FOR mv_i := 1 TO MOVER_NUMBER BY 1 DO
    // Only check for bMoverSync when the WaitOnExternalTrigger scenario is selected
    IF __ISVALIDREF(_MoverList[mv_i].Station.Process) AND
       _MoverList[mv_i].Station.ApproachScenario = ApproachScenario_e.WaitOnExternalTrigger THEN
        //bMoverSync := bMoverSync AND
        //              (_MoverList[i].Station.Process.xMoverPathFree AND NOT _MoverList[i].Station.Process.xNeedMover);
    END_IF
END_FOR

// start update simu mover **********************************************
IF CONST.USE_SIMULATION THEN
    FOR mv_i := 1 TO MOVER_NUMBER BY 1 DO
        _MoverList[mv_i].MoverAxis(xIN_StopMover := HMI_xStopMover);
    END_FOR
END_IF

// stop update simu mover **********************************************

// start communication with B&R PLC ************************************
FOR mv_i := 1 TO CONST.STATION_NUMBER BY 1 DO
    IF __ISVALIDREF(_MoverList[mv_i].Station) AND __ISVALIDREF(_20_AUTO.recipe) THEN
        _StationList[mv_i].Offset := _20_AUTO.recipe.stationOffsets[mv_i - 1];
    END_IF
END_FOR

IF CONST.BIND_WITH_TRACK AND gMoverAxis.Q_CT_Track_to_BR.asStruct.bCommand.enableProcess THEN
    FOR mv_i := 1 TO MOVER_NUMBER BY 1 DO
        IF __ISVALIDREF(_MoverList[mv_i].Station) THEN
            gMoverAxis.Q_CT_Shuttle_to_BR.asStruct[mv_i].bCommand.release :=
                ((THIS^._MoverList[mv_i].State = MoverState_e.WaitLeaveCurrentStation) OR
                (_MoverList[mv_i].State = MoverState_e.MovingToStation) OR
                (_MoverList[mv_i].State = MoverState_e.PerformRelativeMove)) AND
                gMoverAxis.I_CT_Shuttle_from_BR.asStruct[mv_i].bStatus.at_target;

            gMoverAxis.Q_CT_Shuttle_to_BR.asStruct[mv_i].bNextStation    := _MoverList[mv_i].Station.SuperTrackNumber;
            gMoverAxis.Q_CT_Shuttle_to_BR.asStruct[mv_i].diNextOffset_um :=
                LREAL_TO_DINT(_MoverList[mv_i].Station.Offset * 1000.0 +
                              _MoverList[mv_i].MovingProcessOffset * 1000.0);

            // echo At_Target
            gMoverAxis.Q_CT_Shuttle_to_BR.asStruct[mv_i].bCommand.echo_At_Target :=
                gMoverAxis.I_CT_Shuttle_from_BR.asStruct[mv_i].bStatus.at_target;

            // echo at position
            gMoverAxis.Q_CT_Shuttle_to_BR.asStruct[mv_i].bCommand.echo_in_pos :=
                gMoverAxis.I_CT_Shuttle_from_BR.asStruct[mv_i].bStatus.in_position;

            // Quit
            gMoverAxis.Q_CT_Track_to_BR.asStruct.bCommand.resetErrors := HMI.btArMain[7].press;
        END_IF
    END_FOR
END_IF

// stop communication with B&R PLC ************************************

// test if path is free
IF CONST.BIND_WITH_TRACK THEN
    gMoverAxis.Q_CT_Track_to_BR.asStruct.bCommand.wholePathFree := TRUE;

    FOR mv_i := 1 TO CONST.STATION_NUMBER BY 1 DO
        IF __ISVALIDREF(_StationList[mv_i].Process) AND_THEN NOT _StationList[mv_i].Process.xMoverPathFree THEN
            gMoverAxis.Q_CT_Track_to_BR.asStruct.bCommand.wholePathFree := FALSE;
        END_IF
    END_FOR

    IF HMI.enState = enState.StateMANU THEN
        gMoverAxis.Q_CT_Track_to_BR.asStruct.bCommand.wholePathFree := TRUE;
    END_IF
END_IF

// start collision check **********************************************
IF NOT CONST.BIND_WITH_TRACK THEN
    FOR mv_i := 1 TO MOVER_NUMBER - 1 BY 1 DO
        _MoverList[mv_i].MoverAxis.IsColliding(_MoverList[mv_i + 1].MoverAxis);
        _MoverList[mv_i].MoverAxis.WillCollide(_MoverList[mv_i + 1].MoverAxis);

        IF THIS^.IsMoverLost(THIS^._MoverList[mv_i]) THEN
            // ASSERT HERE, WE SHOULD NEVER GO HERE
            ASSERT(0);
        END_IF
    END_FOR

    _MoverList[MOVER_NUMBER].MoverAxis.IsColliding(_MoverList[1].MoverAxis); // do not forget to test this case, too
    _MoverList[MOVER_NUMBER].MoverAxis.WillCollide(_MoverList[1].MoverAxis);
END_IF

// end collision check **********************************************

// start output affectation **********************************************
xOUT_AllMoverEmpty := TRUE;

FOR mv_i := 1 TO MOVER_NUMBER BY 1 DO
    IF _MoverList[mv_i].GetLastStationDone() <> 0 THEN
        xOUT_AllMoverEmpty := FALSE;
    END_IF
END_FOR

xOUT_Error := gMoverAxis.I_CT_Track_from_BR.asStruct.bStatus.error;

// end output affectation **********************************************

// This method check if the wait pos of a given station is before another
// station. This situation is not permitted by the system, yet
METHOD CheckWaitPosNotBehindStation : BOOL
VAR_INPUT
END_VAR
VAR
    i : INT;
END_VAR
CheckWaitPosNotBehindStation := FALSE;
FOR i := 2 TO CONST.STATION_NUMBER BY 1 DO
    CheckWaitPosNotBehindStation := CheckWaitPosNotBehindStation OR
        THIS^._StationList[i].Position.lrWorkPosition + THIS^._StationList[i].WaitPos <
        THIS^._StationList[i - 1].Position.lrWorkPosition;
END_FOR

// NO CHECK ARE MADE BETWEEN THE FIRST POS AND THE LAST
END_METHOD

METHOD Equals : BOOL
VAR_INPUT
    object : ANY;
END_VAR
Equals := THIS = object.pValue;
END_METHOD

METHOD FB_init : BOOL
VAR_INPUT
    bInitRetains : BOOL; // if TRUE, the retain variables are initialized (warm start / cold start)
    bInCopyCode  : BOOL; // if TRUE, the instance afterwards gets moved into the copy code (online change)
END_VAR
VAR
    i : INT;
END_VAR
THIS^._iID := THIS^._iInstanceCounter;
THIS^._iInstanceCounter := THIS^._iInstanceCounter +1;
END_METHOD

METHOD GetMoverIndex : INT
VAR_INPUT
    mover : REFERENCE TO FB_Mover;
END_VAR
VAR
    i : INT;
END_VAR
FOR i:= 1 TO THIS^.MOVER_NUMBER BY 1 DO 
	IF mover.Equals(THIS^._MoverList[i]) THEN
		GetMoverIndex := i;
		EXIT;
	END_IF
END_FOR
END_METHOD

// Get the mover with the next number (Means the mover behind)
METHOD GetNextMover : REFERENCE TO FB_Mover
VAR_INPUT
    Mover : REFERENCE TO FB_Mover;
END_VAR
VAR
    moverIndex : INT;
END_VAR
moverIndex := THIS^.GetMoverIndex(Mover);

IF moverIndex >= THIS^.MOVER_NUMBER THEN
    GetNextMover REF= THIS^._MoverList[1];
ELSE
    GetNextMover REF= THIS^._MoverList[moverIndex + 1];
END_IF
END_METHOD

// we check if there is a mover between refMover and the refMover.Station
// This method is used to unblock a mover that cannot move because of a mover
// "Behind" it that also want to move to the same station
METHOD PRIVATE GetNumOfMoverOnTheWay : INT
VAR_INPUT
    refMover : REFERENCE TO FB_Mover; // The maybe stucking mover
END_VAR
VAR
    lrMoverPosTemp   : LREAL; // we use this position beacuse maybe we are at the end of the track
    lrStationPosTemp : LREAL; // we use this position beacuse maybe we are at the end of the track
    i                : INT;
END_VAR
GetNumOfMoverOnTheWay := 0;

FOR i := 1 TO THIS^.MOVER_NUMBER BY 1 DO
    // If the mover is in front of the tested mover, we add MAX_TRACK_LENGTH (maybe we are at the end of the track ?)
    IF refMover.IsInFront(THIS^._MoverList[i].MoverAxis.CurrentPos) THEN
        lrMoverPosTemp := THIS^._MoverList[i].MoverAxis.CurrentPos + CONST.MAX_TRACK_LENGTH;
    ELSE
        lrMoverPosTemp := THIS^._MoverList[i].MoverAxis.CurrentPos;
    END_IF

    // If the mover is in front of the station, we add MAX_TRACK_LENGTH (maybe we are at the end of the track ?)
    IF refMover.IsInFront(refMover.Station.Position.lrWorkPosition) THEN
        lrStationPosTemp := refMover.Station.Position.lrWorkPosition + CONST.MAX_TRACK_LENGTH;
    ELSE
        lrStationPosTemp := refMover.Station.Position.lrWorkPosition;
    END_IF

    IF (lrMoverPosTemp > refMover.MoverAxis.CurrentPos) AND
       (lrMoverPosTemp <= lrStationPosTemp + refMover.AttachedPieceHolder.PosOffset) THEN
	   // If a mover is at position but has
        GetNumOfMoverOnTheWay := GetNumOfMoverOnTheWay + 1;
    END_IF
END_FOR
END_METHOD

// Get the mover with the previous number (Means the front mover)
METHOD GetPrevMover : REFERENCE TO FB_Mover
VAR_INPUT
    Mover : REFERENCE TO FB_Mover;
END_VAR
VAR
    moverIndex : INT;
END_VAR
moverIndex := THIS^.GetMoverIndex(Mover);

IF moverIndex <= 1 THEN
    GetPrevMover REF= THIS^._MoverList[THIS^.MOVER_NUMBER];
ELSE
    GetPrevMover REF= THIS^._MoverList[moverIndex - 1];
END_IF
END_METHOD

METHOD IsAllMoverAtPosition : BOOL
VAR_INPUT
END_VAR
VAR
    i : INT;
END_VAR
IsAllMoverAtPosition := TRUE;

FOR i := 1 TO THIS^.MOVER_NUMBER BY 1 DO
    IF (THIS^._MoverList[i].State = MoverState_e.WaitLeaveCurrentStation) OR
       (THIS^._MoverList[i].State = MoverState_e.MovingToStation) OR
       (THIS^._MoverList[i].State = MoverState_e.InStationPos) THEN
        IsAllMoverAtPosition := FALSE;
        EXIT;
    END_IF
END_FOR
END_METHOD

// Is a shuttle present in the given region?
// If 'from_pos' is greater than 'to_pos', this means we look in
// a region that include the begining of the track
METHOD PUBLIC IsMoverInRange : BOOL
VAR_INPUT
    from_pos : LREAL; // begin of the tested region (included)
    to_pos   : LREAL; // end of the tested region (included)
END_VAR
VAR
    i       : INT;
END_VAR

IsMoverInRange := FALSE;

IF from_pos < to_pos THEN
    FOR i := 1 TO THIS^.MOVER_NUMBER BY 1 DO
        IF (THIS^._MoverList[i].MoverAxis.CurrentPos >= from_pos) AND
           (THIS^._MoverList[i].MoverAxis.CurrentPos <= to_pos) THEN
		   IsMoverInRange := TRUE;
		   EXIT;
		   
        END_IF
    END_FOR
ELSE // we test a region that pass by the maximum track length
    FOR i := 1 TO THIS^.MOVER_NUMBER BY 1 DO
        IF (THIS^._MoverList[i].MoverAxis.CurrentPos >= from_pos) OR
           (THIS^._MoverList[i].MoverAxis.CurrentPos <= to_pos) THEN
		   IsMoverInRange := TRUE;
		   EXIT;
		   
        END_IF
    END_FOR
END_IF
END_METHOD

// If the target station of a mover is not between the target of the previous and the next mover
// this function will return true. This function is attendend to debug only
METHOD IsMoverLost : BOOL
VAR_INPUT
    mover : REFERENCE TO FB_Mover;
END_VAR
VAR
    i : INT;

    prevStationLoc  : LREAL;
    nextStationLoc  : LREAL;
    moverStationLoc : LREAL; // mover to test location
    posList         : ARRAY[0..2] OF LREAL;
END_VAR
(* the algorithm function as fallow 

First we built a sorted array based on the station position
Then we search for the previous station position and fix
our search index
Then we check if the squence of mover is correct. The sequence must be
PreviousMoverStation -> CurrentMoverStation -> NextMoverStation
If we don't get this sequence, then the mover is lost.

In fact, since we have only 3 elements, we only need to check
the next station
*)
IsMoverLost := FALSE;

nextStationLoc  := THIS^.GetNextMover(mover).Station.Position.lrWorkPosition;
prevStationLoc  := THIS^.GetPrevMover(mover).Station.Position.lrWorkPosition;
moverStationLoc := mover.station.Position.lrWorkPosition;

posList[0] := prevStationLoc;
posList[1] := moverStationLoc;
posList[2] := nextStationLoc;

SortBubbleLREAL(ADR(posList), 0, 2);

IF posList[0] = prevStationLoc THEN
    IF posList[1] <> moverStationLoc THEN
        IsMoverLost := TRUE;
    END_IF

ELSIF posList[0] = moverStationLoc THEN
    IF posList[1] <> nextStationLoc THEN
        IsMoverLost := TRUE;
    END_IF

ELSE (* posList[0] = nextStationLoc *)
    IF posList[1] <> prevStationLoc THEN
        IsMoverLost := TRUE;
    END_IF
END_IF
END_METHOD

METHOD PRIVATE IsMoverMovingToStation : BOOL
VAR_INPUT
    iMoverNumber : INT; // the current mover number 
END_VAR
VAR
    i           : INT;
END_VAR
IsMoverMovingToStation := FALSE;

FOR i := 1 TO THIS^.MOVER_NUMBER BY 1 DO

    // we don't check the tests mover station, else it will be always true
    IF (iMoverNumber <> i) AND THIS^._MoverList[i].Station.Equals(THIS^._MoverList[iMoverNumber].Station) THEN
        IsMoverMovingToStation := IsMoverMovingToStation OR
                                  (THIS^._MoverList[i].State = MoverState_e.WaitLeaveCurrentStation) OR
                                  (THIS^._MoverList[i].State = MoverState_e.MovingToStation) OR
                                  (THIS^._MoverList[i].State = MoverState_e.InStationPos);

        // Do not exit here, since we OR the flag
        // TODO maybe we should add an IF statement to exit when the flag is true
        // because it will never be false again ... ? // PERFORMANCE ISSUE
    END_IF

END_FOR
END_METHOD

// Return TRUE if at least one mover is stucked
METHOD IsMoverStucked : BOOL
VAR_INPUT
END_VAR
IsMoverStucked := FALSE;

FOR mv_i := 1 TO THIS^.MOVER_NUMBER BY 1 DO
    IF THIS^._MoverList[mv_i].MoverAxis.xStuck THEN
        IsMoverStucked := TRUE;
        EXIT;
    END_IF
END_FOR
END_METHOD

// Is the given process used by the current station configuration?
METHOD IsProcessUsed : BOOL
VAR_INPUT
    this_process : REFERENCE TO FB_AUT_ABSTRACT;
END_VAR
VAR
	i : INT;
END_VAR
IsProcessUsed := THIS^._WorkStationList[PH_num].IsProcessUsed(this_process);
END_METHOD

METHOD SetAllScenario : REFERENCE TO FB_MoverMan
VAR_INPUT
END_VAR
VAR
	i : INT;
END_VAR
FOR i := 1 TO CONST.STATION_NUMBER BY 1 DO
    THIS^._StationList[i].ApproachScenario := THIS^.HMI_Scenario;
END_FOR

SetAllScenario REF= THIS^;
END_METHOD

// Give a random time for each process. It ensure at least the minimum and the maximum value are given
// to at least 2 diffrents process
METHOD SetAllTimers : REFERENCE TO FB_MoverMan
VAR_INPUT
    arrStationTime : POINTER TO DINT;
    udiOffset      : UDINT; // simple offset to apply to the seed
END_VAR
VAR
    i         : INT;
    rand      : DRAND;
    tempIndex : INT := 0;
    getTime   : GETSYSTEMTIME;
END_VAR
IF arrStationTime <> 0 THEN
	
    getTime();
    rand.Seed := TO_INT(getTime.timeLoDW + udiOffset);

    FOR i := 0 TO CONST.STATION_NUMBER - 1 BY 1 DO
        rand();
        arrStationTime[i] := TO_DINT((THIS^.HMI_TimeMax - THIS^.HMI_TimeMin) * (rand.Num) + THIS^.HMI_TimeMin);
    END_FOR

    tempIndex := 0;

    FOR i := 1 TO CONST.STATION_NUMBER - 1 BY 1 DO
        IF arrStationTime[i] < arrStationTime[tempIndex] THEN
            tempIndex := i;
        END_IF
    END_FOR

    arrStationTime[tempIndex] := THIS^.HMI_TimeMin;

    tempIndex := 0;

    FOR i := 1 TO CONST.STATION_NUMBER - 1 BY 1 DO
        IF arrStationTime[i] > arrStationTime[tempIndex] THEN
            tempIndex := i;
        END_IF
    END_FOR

    arrStationTime[tempIndex] := THIS^.HMI_TimeMax;
END_IF

SetAllTimers REF= THIS^;
END_METHOD

METHOD ToString : STRING
VAR_INPUT
END_VAR
ToString := CONCAT('FB_MoverMan_', TO_STRING(THIS^._iID));
END_METHOD

END_FUNCTION_BLOCK

// ---- POUs/20_AUTO/Mover/FB_PieceHolder.TcPOU
FUNCTION_BLOCK FB_PieceHolder
VAR_INPUT
END_VAR
VAR_OUTPUT
END_VAR
VAR
	_lrPosOffset : LREAL; // current offset position
	
	_iID : INT := 0; // instance ID, is set during FB_Init using the value of _iInstanceCounter 
END_VAR
VAR_STAT
	_iInstanceCounter : INT := 1; // instance counter
END_VAR

METHOD FB_init : BOOL
VAR_INPUT
    bInitRetains : BOOL;  // if TRUE, the retain variables are initialized (warm start / cold start)
    bInCopyCode  : BOOL;  // if TRUE, the instance afterwards gets moved into the copy code (online change)
    offset       : LREAL; //position offset of the tool using this toolhead, a negative value represents a move on the left
END_VAR
THIS^._iID := THIS^._iInstanceCounter;
THIS^._iInstanceCounter := THIS^._iInstanceCounter +1;
THIS^.PosOffset := offset;
END_METHOD

PROPERTY PosOffset : LREAL
GET
PosOffset := _lrPosOffset;
END_GET
SET
_lrPosOffset := PosOffset;
END_SET
END_PROPERTY

METHOD ToString : STRING
VAR_INPUT
END_VAR
ToString := CONCAT('FB_PieceHolder_', TO_STRING(THIS^._iID));
END_METHOD

END_FUNCTION_BLOCK

// ---- POUs/20_AUTO/Mover/FB_SimuMoverAxis.TcPOU
FUNCTION_BLOCK FB_SimuMoverAxis IMPLEMENTS IObject
VAR_INPUT
    xIN_StopMover : BOOL; // stop the mover from movinf
END_VAR
VAR_OUTPUT
    outSimuCurrentPos   : Pos2D_t; // Mover position, expressed as slot number
    outSimuCurrentPosSC : Pos2D_t; // Mover position, expressed as pixel for SC
    outSimuCurrentRot   : INT;     // mover current rotation
    isInPos             : BOOL;    // true when targetPos = currentPos
END_VAR
VAR
    // with tick rate at 10ms, a value of 10 gives us 1m/s
    _Velocity    : LREAL := 0;     // Mover velocity, expressed as mm per tick, max is 10m/s
    _ErrorState  : INT   := 0;     // error state, not used
    _TargetPos   : LREAL := 0;     // last target pos
    _CurrentPos  : LREAL := 0;     // Current Pos, but with more resolution than the pixel
    _IsColliding : BOOL  := FALSE; // When true, the mover should not move
    _LastPos     : LREAL := 0;     // last position, used to trigger the xStuck flag
    _xStuck      : BOOL;           // true when the axis does not move
    _willCollide : BOOL := FALSE;  // TRUE if a collision will occure with the current velocity

    {attribute 'hide'}
    _lrNextStopPos : LREAL; // local variable used to get next stop

    _iID : INT := 0; // instance ID, is set during FB_Init using the value of _iInstanceCounter 

    _CurrentDir : MoverDirection_e := MoverDirection_e.Farward;
END_VAR

VAR_TEMP
    _MoverAccel : LREAL; // Mover acceleration, can be positive or negative depending on the direction
END_VAR

VAR CONSTANT
    MAX_POS  : LREAL := CONST.MAX_TRACK_LENGTH; // should be defined elsewhere ...
    MAX_SIZE : LREAL := CONST.MAX_MOVER_SIZE;   // Maxium size of the mover
    //MOVER_ACCEL        : LREAL := 0.1;                      // Mover acceleration, in mm/tick^2
    //MOVER_VELOCITY_MAX : LREAL := 20;                     // Mover velocity, expressed as mm per tick, max is 10m/s
    MOVER_VELOCITY_MIN : LREAL := 1; // Mover velocity, expressed as mm per tick, max is 10m/s
END_VAR
VAR_STAT
    _iInstanceCounter : INT := 1; // instance counter
END_VAR

IF NOT xIN_StopMover THEN // Do not change momemtum when we stop the movers from HMI
    IF MoverDirection_e.Farward = THIS^._CurrentDir THEN
        _MoverAccel := SIMU.lrAccelMover;
    ELSE
        _MoverAccel := -SIMU.lrAccelMover;
    END_IF

    IF NOT _IsColliding THEN

        IF THIS^.GetStopLen(_Velocity, SIMU.lrAccelMover) >= DistToTravel(_CurrentPos, _TargetPos) OR
           THIS^._willCollide THEN
            _Velocity := _Velocity - _MoverAccel;

        ELSIF SIMU.lrSpeedMover > ABS(_Velocity) AND _CurrentPos <> _TargetPos THEN
            _Velocity := _Velocity + _MoverAccel;

        END_IF
    ELSE
        _Velocity := _Velocity - _MoverAccel;
    END_IF
END_IF

// protect max and min speed
IF SIMU.lrSpeedMover < ABS(_Velocity) THEN
    IF MoverDirection_e.Farward = THIS^._CurrentDir THEN
        _Velocity := SIMU.lrSpeedMover;
    ELSE
        _Velocity := -SIMU.lrSpeedMover;
    END_IF
ELSIF ABS(_Velocity) < MOVER_VELOCITY_MIN THEN
    IF MoverDirection_e.Farward = THIS^._CurrentDir THEN
        _Velocity := MOVER_VELOCITY_MIN;
    ELSE
        _Velocity := -MOVER_VELOCITY_MIN;
    END_IF
END_IF

IF NOT _IsColliding AND NOT xIN_StopMover THEN

    IF DistToTravel(_CurrentPos, _TargetPos) > ABS(_Velocity) THEN
        _CurrentPos := _CurrentPos + _Velocity;

    ELSE
        _CurrentPos := _TargetPos;
        _Velocity   := 0;

    END_IF
END_IF

IF _CurrentPos >= MAX_POS THEN
    _CurrentPos := _CurrentPos - MAX_POS;
    // we prevent the stuck flag to be true at the end of the track
    THIS^._LastPos := THIS^._LastPos - MAX_POS;
END_IF

isInPos := EqualDelta(_CurrentPos, _TargetPos, 1.0); // we use delta comparison beacause axis is always at a low value 

outSimuCurrentPos   := THIS^.ResolvePos(THIS^.CurrentPos, outSimuCurrentRot);
outSimuCurrentPosSC := THIS^.ResolvePosSC(THIS^.CurrentPos, outSimuCurrentRot);

_xStuck        := (THIS^._CurrentPos < (THIS^._LastPos + _Velocity)) AND NOT isInPos;
THIS^._LastPos := THIS^._CurrentPos;

PROPERTY CurrentPos : LREAL
GET
IF CONST.BIND_WITH_TRACK THEN
    CurrentPos := TO_LREAL(gMoverAxis.I_CT_Shuttle_from_BR.asStruct[THIS^._iID].diCurrentPos_um) / 1000.0;
ELSE
    CurrentPos := _CurrentPos;
END_IF
END_GET
SET
END_SET
END_PROPERTY

PROPERTY CurrentVelocity : LREAL
GET
CurrentVelocity := THIS^._Velocity;
END_GET
SET
END_SET
END_PROPERTY

METHOD Equals : BOOL
VAR_INPUT
    object : ANY;
END_VAR
Equals := THIS = object.pValue;
END_METHOD

METHOD FB_init : BOOL
VAR_INPUT
    bInitRetains : BOOL; // if TRUE, the retain variables are initialized (warm start / cold start)
    bInCopyCode  : BOOL; // if TRUE, the instance afterwards gets moved into the copy code (online change)

    PosInit : LREAL; // initial position at startup
END_VAR
THIS^._iID := THIS^._iInstanceCounter;
THIS^._iInstanceCounter := THIS^._iInstanceCounter +1;
IF PosInit < THIS^.MAX_POS THEN
    THIS^._CurrentPos := PosInit;
ELSE
    THIS^._CurrentPos := 0;
END_IF
END_METHOD

METHOD PRIVATE GetStopLen : LREAL
VAR_INPUT
    currentVelocity : LREAL;
    currentAccel    : LREAL;
END_VAR
VAR
    tickToStop : INT;
END_VAR
// This function search the position we will get if we stop now
//
// (velocity)
//     ^          _________   <- we are here, at the end of the top slope
//     |        /          \
//     |       /            \
//     |   ___/              \______
//     |     
//     ┼------------------------------>  (time)
//
// (position)
//     ^ 
//     |                      _________
//     |                  .../
//     |               ../    ^
//     |            ../       |
//     |          ../         we search this position
//     |   ___.../
//     | 
//     ┼------------------------------>  (time)

IF currentAccel <= 0 THEN
    ASSERT(currentAccel > 0);
    RETURN;
END_IF

// TO_INT floor the result, and we need at least 1 tick to stop
tickToStop := TO_INT(currentVelocity / currentAccel) + 1;

GetStopLen := tickToStop * currentVelocity / 2;
END_METHOD

// only check the collision in one way, this prevent
// all the mover chain to be stucked
METHOD IsColliding : BOOL
VAR_INPUT
    nextMover : REFERENCE TO FB_SimuMoverAxis;
END_VAR
IsColliding := FALSE;

IF DistToTravel(THIS^.CurrentPos, nextMover.CurrentPos) <= CONST.MAX_MOVER_SIZE THEN
    IsColliding := TRUE;

END_IF

THIS^._IsColliding := IsColliding;
END_METHOD

METHOD PUBLIC MoveTo : REFERENCE TO FB_SimuMoverAxis
VAR_INPUT
    Position : LREAL; // move the axis to this position
END_VAR
THIS^._TargetPos := Position;
THIS^._CurrentDir := MoverDirection_e.Farward;
isInPos := THIS^._CurrentPos = THIS^._TargetPos;
MoveTo REF= THIS^;
END_METHOD

METHOD ResolvePos : Pos2D_t
VAR_INPUT
    inX      : LREAL;
    rotation : REFERENCE TO INT;
END_VAR
VAR CONSTANT
    (* The track has this dimension in reality
              __________
     1030mm (___________) 1030 mm
              4000 mm
			  
     and we map it like that:
	   __   80 (radius)
	  |  |
	  |  |  800
	  |  |
	  |__|
	        80 (raidus)
    *)
    START_X     : DINT  := 0;
    START_Y     : DINT  := 0;
    MAX_SIMU_DX : DINT  := 120;
    MAX_SIMU_DY : DINT  := 800;
    RADIUS_X    : LREAL := 60.0;
    RADIUS_Y    : LREAL := 100.0;

    FIRST_RADIUS_START  : LREAL := 4000;
    FIRST_RADIUS_END    : LREAL := 5030;
    SECOND_RADIUS_START : LREAL := 9030;
    SECOND_RADIUS_END   : LREAL := 10060;
END_VAR

VAR
    x_rad_calc : LREAL;
    y_rad_calc : LREAL;
    FACTOR_Y   : LREAL;
END_VAR
FACTOR_Y := FIRST_RADIUS_START / MAX_SIMU_DY;

IF inX < 0 THEN
    ResolvePos.x := START_X;
    ResolvePos.y := START_Y;
    rotation     := 0;

ELSIF inX >= 0 AND inX <= FIRST_RADIUS_START THEN
    ResolvePos.x := START_X;
    ResolvePos.y := START_Y + TO_DINT(inX / FACTOR_Y);
    rotation     := 0;

ELSIF inX > FIRST_RADIUS_START AND inX < FIRST_RADIUS_END THEN

    // should go between -1RAD and +1RAD
    x_rad_calc   := ((inX - FIRST_RADIUS_START) * 2 / (FIRST_RADIUS_END - FIRST_RADIUS_START) - 1) * PI / 2;
    ResolvePos.x := TO_DINT(SIN(x_rad_calc) * RADIUS_X) + START_X + TO_DINT(RADIUS_X);

    // should go from 0RAD to 1RAD, then 0RAD
    y_rad_calc   := (1 - (inX - FIRST_RADIUS_START) * 2 / (FIRST_RADIUS_END - FIRST_RADIUS_START)) * PI / 2;
    ResolvePos.y := TO_DINT(COS(y_rad_calc) * RADIUS_Y + START_Y + MAX_SIMU_DY);

    rotation := TO_INT(SIN(x_rad_calc) * 90 + 90);

ELSIF inX >= FIRST_RADIUS_END AND inX <= SECOND_RADIUS_START THEN
    ResolvePos.x := START_X + MAX_SIMU_DX;
    ResolvePos.y := START_Y + MAX_SIMU_DY - TO_DINT((inX - FIRST_RADIUS_END) / FACTOR_Y);
    rotation     := 180;

ELSIF inX > SECOND_RADIUS_START AND inX < SECOND_RADIUS_END THEN
    // should go between -1RAD and +1RAD
    x_rad_calc   := ((inX - SECOND_RADIUS_START) * 2 / (SECOND_RADIUS_END - SECOND_RADIUS_START) - 1) * PI / 2;
    ResolvePos.x := START_X - TO_DINT(SIN(x_rad_calc) * RADIUS_X) + TO_DINT(RADIUS_X);

    // should go from 0RAD to 1RAD, then 0RAD
    y_rad_calc   := (1 - (inX - SECOND_RADIUS_START) * 2 / (SECOND_RADIUS_END - SECOND_RADIUS_START)) * PI / 2;
    ResolvePos.y := START_Y - TO_DINT(COS(y_rad_calc) * RADIUS_Y);

    rotation := TO_INT(SIN(x_rad_calc) * 90 + 270);

ELSE
    ResolvePos.x := START_X;
    ResolvePos.y := START_Y;
    rotation     := 0;

END_IF
END_METHOD

METHOD ResolvePosSC : Pos2D_t
VAR_INPUT
    inX      : LREAL;
    rotation : REFERENCE TO INT;
END_VAR
VAR CONSTANT
    (* The track has this dimension in reality
              __________
     1030mm (___________) 1030 mm
              4000 mm
			  
     and we map it like that:
	   __   80 (radius)
	  |  |
	  |  |  800
	  |  |
	  |__|
	        80 (raidus)
    *)
    START_X     : DINT  := 0;
    START_Y     : DINT  := 0;
    MAX_SIMU_DX : DINT  := 70;
    MAX_SIMU_DY : DINT  := 800;
    RADIUS_X    : LREAL := 35;
    RADIUS_Y    : LREAL := 65.0;

    FIRST_RADIUS_START  : LREAL := 4000;
    FIRST_RADIUS_END    : LREAL := 5030;
    SECOND_RADIUS_START : LREAL := 9030;
    SECOND_RADIUS_END   : LREAL := 10060;
END_VAR

VAR
    x_rad_calc : LREAL;
    y_rad_calc : LREAL;
    FACTOR_Y   : LREAL;
END_VAR
FACTOR_Y := FIRST_RADIUS_START / MAX_SIMU_DY;

IF inX < 0 THEN
    ResolvePosSC.x := START_X;
    ResolvePosSC.y := START_Y;
    rotation       := 0;

ELSIF inX >= 0 AND inX <= FIRST_RADIUS_START THEN
    ResolvePosSC.x := START_X;
    ResolvePosSC.y := START_Y + TO_DINT(inX / FACTOR_Y);
    rotation       := 0;

ELSIF inX > FIRST_RADIUS_START AND inX < FIRST_RADIUS_END THEN

    // should go between -1RAD and +1RAD
    x_rad_calc     := ((inX - FIRST_RADIUS_START) * 2 / (FIRST_RADIUS_END - FIRST_RADIUS_START) - 1) * PI / 2;
    ResolvePosSC.x := TO_DINT(SIN(x_rad_calc) * RADIUS_X) + START_X + TO_DINT(RADIUS_X);

    // should go from 0RAD to 1RAD, then 0RAD
    y_rad_calc     := (1 - (inX - FIRST_RADIUS_START) * 2 / (FIRST_RADIUS_END - FIRST_RADIUS_START)) * PI / 2;
    ResolvePosSC.y := TO_DINT(COS(y_rad_calc) * RADIUS_Y + START_Y + MAX_SIMU_DY);

    rotation := TO_INT(SIN(x_rad_calc) * 90 + 90);

ELSIF inX >= FIRST_RADIUS_END AND inX <= SECOND_RADIUS_START THEN
    ResolvePosSC.x := START_X + MAX_SIMU_DX;
    ResolvePosSC.y := START_Y + MAX_SIMU_DY - TO_DINT((inX - FIRST_RADIUS_END) / FACTOR_Y);
    rotation       := 180;

ELSIF inX > SECOND_RADIUS_START AND inX < SECOND_RADIUS_END THEN
    // should go between -1RAD and +1RAD
    x_rad_calc     := ((inX - SECOND_RADIUS_START) * 2 / (SECOND_RADIUS_END - SECOND_RADIUS_START) - 1) * PI / 2;
    ResolvePosSC.x := START_X - TO_DINT(SIN(x_rad_calc) * RADIUS_X) + TO_DINT(RADIUS_X);

    // should go from 0RAD to 1RAD, then 0RAD
    y_rad_calc     := (1 - (inX - SECOND_RADIUS_START) * 2 / (SECOND_RADIUS_END - SECOND_RADIUS_START)) * PI / 2;
    ResolvePosSC.y := START_Y - TO_DINT(COS(y_rad_calc) * RADIUS_Y);

    rotation := TO_INT(SIN(x_rad_calc) * 90 + 270);

ELSE
    ResolvePosSC.x := START_X;
    ResolvePosSC.y := START_Y;
    rotation       := 0;

END_IF

ResolvePosSC.x := -ResolvePosSC.x;
END_METHOD

METHOD ToString : STRING
VAR_INPUT
END_VAR
VAR
END_VAR
ToString := CONCAT('FB_SimuMoverAxis_', TO_STRING(THIS^._iID));
END_METHOD

// Use this method in a collider manager so the simu axis 
// will know when to stop itself
METHOD WillCollide : BOOL
VAR_INPUT
    nextMover : REFERENCE TO FB_SimuMoverAxis;
END_VAR
VAR
    diffVelocity : LREAL;
END_VAR
THIS^._willCollide := FALSE;
diffVelocity       := 0;

// If the 2 movers are moving tarwards each other
IF (THIS^._Velocity > 0) AND (nextMover.CurrentVelocity < 0) THEN
    diffVelocity := SQRT(THIS^._Velocity * THIS^._Velocity + (nextMover.CurrentVelocity * nextMover.CurrentVelocity));

    // If the 2 movers are moving in the same direction
ELSE
    IF ABS(THIS^._Velocity) > ABS(nextMover.CurrentVelocity) THEN
        diffVelocity :=
            SQRT(THIS^._Velocity * THIS^._Velocity - (nextMover.CurrentVelocity * nextMover.CurrentVelocity));
    END_IF
END_IF

THIS^._willCollide
    := DistToTravel(THIS^.CurrentPos, nextMover.CurrentPos) <=
       THIS^.GetStopLen(diffVelocity, SIMU.lrAccelMover) + CONST.MAX_MOVER_SIZE;

WillCollide := THIS^._willCollide;
END_METHOD

PROPERTY xStuck : BOOL
GET
xStuck := _xStuck;
END_GET
SET
END_SET
END_PROPERTY

END_FUNCTION_BLOCK

// ---- POUs/20_AUTO/Mover/DistToTravel.TcPOU
// Get the distance to travel from startPos to stopPos
FUNCTION DistToTravel : LREAL
VAR_INPUT
    startPos : LREAL;
    stopPos  : LREAL;
END_VAR
VAR
END_VAR

IF startPos > stopPos THEN
    DistToTravel := stopPos - startPos + CONST.MAX_TRACK_LENGTH;
ELSE
    DistToTravel := stopPos - startPos;
END_IF

END_FUNCTION

// ---- POUs/20_AUTO/TOOL/ASSERT.TcPOU
FUNCTION ASSERT : BOOL
VAR_INPUT
    bStatement : BOOL; // Should be true, else raise an error
END_VAR
VAR
END_VAR

IF NOT  bStatement THEN
	ASSERT := TRUE;
ELSE
	ASSERT := FALSE;
END_IF

END_FUNCTION

// ---- POUs/20_AUTO/Mover/FB_Mover.TcPOU
FUNCTION_BLOCK FB_Mover IMPLEMENTS IObject
VAR_INPUT
END_VAR
VAR_OUTPUT
END_VAR
VAR
    _ID           : INT;                           // hard id number of the mover
    _MoverAxis    : REFERENCE TO FB_SimuMoverAxis; // reference to an FB_SimuMoverAxis
    _AttachedTool : REFERENCE TO FB_PieceHolder;   // attached toolhead
    _Station      : REFERENCE TO FB_Station;       // current station

    _State : MoverState_e := MoverState_e.WaitOnNextStation; // current mover state

    _ActualTargetOffset  : LREAL; // final offset to apply to the current/next target
    _MovingProcessOffset : LREAL; (* added offset by the process, 
                                     used to compute the new position of the shuttle inside the station *)

    _LastStationDone : INT;    // the number of the last station done. If negative, the piece is not good at this station
    _ErrorCode       : STRING; // The error code that comes with the last station done. reset afer 

    _iID : INT := 0; // instance ID, is set during FB_Init using the value of _iInstanceCounter 
END_VAR
VAR CONSTANT
END_VAR
VAR_STAT
    _iInstanceCounter : INT := 1; // instance counter
END_VAR

// This is the final offset to apply when moving to a target
PROPERTY PUBLIC ActualTargetOffset : LREAL
GET
ActualTargetOffset := THIS^._ActualTargetOffset;
END_GET
END_PROPERTY

PROPERTY AttachedPieceHolder : REFERENCE TO FB_PieceHolder
GET
AttachedPieceHolder REF=_AttachedTool;
END_GET
SET
_AttachedTool REF= AttachedPieceHolder;
END_SET
END_PROPERTY

METHOD Equals : BOOL
VAR_INPUT
    object : ANY;
END_VAR
Equals := THIS = object.pValue;
END_METHOD

METHOD FB_init : BOOL
VAR_INPUT
    bInitRetains : BOOL; // if TRUE, the retain variables are initialized (warm start / cold start)
    bInCopyCode  : BOOL; // if TRUE, the instance afterwards gets moved into the copy code (online change)
    ID           : INT;  // hard id number of the mover

    MoverAxis : REFERENCE TO FB_SimuMoverAxis; // reference to an FB_SimuMoverAxis
END_VAR
THIS^._iID := THIS^._iInstanceCounter;
THIS^._iInstanceCounter := THIS^._iInstanceCounter +1;
THIS^._ID := ID;
THIS^._MoverAxis REF= MoverAxis;
THIS^._AttachedTool REF=0;
THIS^._Station REF=0;
END_METHOD

METHOD GetErrorCode : STRING
VAR_INPUT
END_VAR
GetErrorCode := THIS^._ErrorCode;
END_METHOD

// Get the last station done. The number is always positive
// To know if the piece is bad, you have to use the IsPieceBad method
METHOD PUBLIC GetLastStationDone : INT
VAR_INPUT
END_VAR
GetLastStationDone := ABS(THIS^._LastStationDone);
END_METHOD

// Is this mover behind a given position?
// this method do the opposit as IsInFront
METHOD IsBehind : BOOL
VAR_INPUT
    lrPosition : LREAL; // position to test
END_VAR
IsBehind := lrPosition > THIS^._MoverAxis.CurrentPos;
END_METHOD

// Is this mover is in front of a given position?
// Use this function also to check if the next station is behind the mover or not.
// In this case, the mover needs to complet its turn for accessing the given station
METHOD IsInFront : BOOL
VAR_INPUT
    lrPosition : LREAL; // position to test
END_VAR
IsInFront := lrPosition < THIS^._MoverAxis.CurrentPos;
END_METHOD

METHOD IsInStationPos : BOOL
VAR_INPUT
END_VAR
// we have to substract the piecholder offset to find the station position again
IF CONST.BIND_WITH_TRACK THEN
    // IsInStationPos :=
    //     THIS^.Station.Position.isInPos(gMoverAxis.I_CT_Shuttle_from_BR.asStruct[THIS^._ID].diCurrentPos_um / 1000 -
    //                                    THIS^._AttachedTool.PosOffset -
    //                                    THIS^.Station.Offset);
    IF __ISVALIDREF(THIS^.Station) THEN
        //IsInStationPos :=
        //    gMoverAxis.I_CT_Shuttle_from_BR.asStruct[THIS^._ID].bStatus.at_target AND
        //    (gMoverAxis.I_CT_Shuttle_from_BR.asStruct[THIS^._ID].bDestinationStation = THIS^.Station.SuperTrackNumber);
        IsInStationPos :=
            THIS^.Station.Position.isInPos(gMoverAxis.I_CT_Shuttle_from_BR.asStruct[THIS^._ID].diCurrentPos_um / 1000 -
                                           THIS^._AttachedTool.PosOffset -
                                           THIS^.Station.Offset -
                                           THIS^._MovingProcessOffset) AND
            gMoverAxis.I_CT_Shuttle_from_BR.asStruct[THIS^._ID].bStatus.at_target;
    ELSE
        IsInStationPos := FALSE;
    END_IF
ELSE
    IsInStationPos := THIS^.Station.Position
        .isInPos(THIS^.MoverAxis.CurrentPos - THIS^._AttachedTool.PosOffset - THIS^.Station.Offset);
END_IF
END_METHOD

// Is the carried piece bad? A piece is bad when the last visited station
// is negative
METHOD PUBLIC IsPieceBad : BOOL
VAR_INPUT
END_VAR
IsPieceBad := THIS^._LastStationDone < 0;
END_METHOD

PROPERTY MoverAxis : REFERENCE TO FB_SimuMoverAxis
GET
MoverAxis REF= _MoverAxis;
END_GET
SET
_MoverAxis REF= MoverAxis;
END_SET
END_PROPERTY

// When a mover is given to a process, this process is allowed to
// use this command to move the shuttle
METHOD PUBLIC MoveRelativeInsideStation : BOOL
VAR_INPUT
    offsetPosition : LREAL;
END_VAR
MoveRelativeInsideStation := FALSE;

IF (MoverState_e.InOperation = THIS^.State) AND
   (ABS(offsetPosition + THIS^.Station.Offset + THIS^._MovingProcessOffset) < LREAL#500.0) THEN
    THIS^.State                := MoverState_e.PerformRelativeMove;
    THIS^._MovingProcessOffset := offsetPosition + THIS^._MovingProcessOffset;
    MoveRelativeInsideStation  := TRUE;
END_IF
END_METHOD

// Move to the current set station. Can only move if the current process are running
METHOD MoveToStation : REFERENCE TO FB_Mover
VAR_INPUT
END_VAR
IF THIS^._State <> MoverState_e.InOperation THEN
    THIS^.MoverAxis
        .MoveTo(TO_POS(THIS^.Station.Position.lrWorkPosition + THIS^._AttachedTool.PosOffset + THIS^.Station.Offset));

    THIS^._MovingProcessOffset := 0;
    THIS^._ActualTargetOffset  := THIS^._AttachedTool.PosOffset + THIS^.Station.Offset;
    THIS^._State               := MoverState_e.WaitLeaveCurrentStation;
ELSE
    ASSERT(0); // should not be called when we are in operation !
END_IF

MoveToStation REF= THIS^;
END_METHOD

// Move to waiting spot
// The mover will not move if the waiting spot can not store
// a full mover
METHOD MoveToWaitSpot : REFERENCE TO FB_Mover
VAR_INPUT
END_VAR
IF THIS^._State <> MoverState_e.InOperation THEN
    IF THIS^.Station.WaitPos <= (THIS^.Station.Position.lrWorkPosition - CONST.MAX_MOVER_SIZE) THEN
        THIS^.MoverAxis.MoveTo(TO_POS(THIS^.Station.WaitPos + THIS^._AttachedTool.PosOffset + THIS^.Station.Offset));
    ELSE
        THIS^.MoverAxis.MoveTo(TO_POS(THIS^.Station.Position.lrWorkPosition +
                                      THIS^._AttachedTool.PosOffset +
                                      THIS^.Station.Offset));
    END_IF

    THIS^._MovingProcessOffset := 0;
    THIS^._ActualTargetOffset  := THIS^._AttachedTool.PosOffset + THIS^.Station.Offset + THIS^.Station._WaitPosOffset;
    THIS^._State               := MoverState_e.WaitLeaveCurrentStation;
ELSE
    ASSERT(0); // never use this command when we are in operation
END_IF

MoveToWaitSpot REF= THIS^;
END_METHOD

PROPERTY PUBLIC MovingProcessOffset : LREAL
GET
MovingProcessOffset := THIS^._MovingProcessOffset;
END_GET
END_PROPERTY

METHOD SetErrorCode : BOOL
VAR_INPUT
	error_code : STRING; // error code in string format
END_VAR
IF LEN(THIS^._ErrorCode) > 0 THEN
    SetErrorCode := FALSE;
ELSE
    THIS^._ErrorCode := error_code;
    SetErrorCode     := TRUE;
END_IF
END_METHOD

// Set the last station visited as soon as you won't redo the process
// again on your piece. It is recommanded to first set the piece as bad
// (negative current station number) as soon as the process has begun,
// then if the process has ended successfuly, you can again set
// the last station visited with the positive current station number.
// This method returns FALSE when the absolute value of the given station
// number is smaller than the current value
// To remove pieces from the shuttle, use the UnloadPieces method
METHOD PUBLIC SetLastStation : BOOL
VAR_INPUT
    value : INT;
END_VAR
IF ABS(value) < ABS(THIS^._LastStationDone) THEN
    SetLastStation := FALSE;
ELSE
    IF THIS^._LastStationDone < 0 THEN
        value := 0 - ABS(value);
    END_IF

    THIS^._LastStationDone := value;
    SetLastStation         := TRUE;
END_IF
END_METHOD

// Set a specic piece holder. This will affect the station position offset
METHOD SetPieceHolder : REFERENCE TO FB_Mover
VAR_INPUT
	pieceHolder : REFERENCE TO FB_PieceHolder;
END_VAR
IF __ISVALIDREF(pieceHolder) THEN
	THIS^._AttachedTool REF=pieceHolder;
END_IF
SetPieceHolder REF= THIS^;
END_METHOD

// Set the next station of the mover. This action does not make the mover moves. 
// First you need to set the station. Then, depending on the station scenario,
// you will run to it when its current process is finished or move to it
// as quick as possible
METHOD SetStation : REFERENCE TO FB_Mover
VAR_INPUT
	Station : REFERENCE TO FB_Station;
END_VAR
IF __ISVALIDREF(Station) AND_THEN (THIS^._State <> MoverState_e.InOperation) THEN
    THIS^._Station REF= Station;
    THIS^._State   := MoverState_e.WaitOnNextStation;
ELSE
    ASSERT(0);
END_IF

SetStation REF= THIS^;
END_METHOD

PROPERTY State : MoverState_e
GET
State := _State;
END_GET
SET
_State := State;
END_SET
END_PROPERTY

PROPERTY Station : REFERENCE TO FB_Station
GET
Station REF=_Station;
END_GET
SET
_Station REF=Station;
END_SET
END_PROPERTY

// take a position and return always a positive integer between 0 and MAX_TRACK_LENGTH
METHOD PRIVATE TO_POS : DINT
VAR_INPUT
	pos : LREAL;
END_VAR
IF pos < 0 THEN
    TO_POS := LREAL_TO_DINT(pos + CONST.MAX_TRACK_LENGTH);

ELSIF pos >= CONST.MAX_TRACK_LENGTH THEN
    TO_POS := LREAL_TO_DINT(pos) MOD LREAL_TO_DINT(CONST.MAX_TRACK_LENGTH);

ELSE
    TO_POS := LREAL_TO_DINT(pos);

END_IF
END_METHOD

METHOD ToString : STRING
VAR_INPUT
END_VAR
ToString := CONCAT('FB_Mover_', TO_STRING(THIS^._iID));
END_METHOD

// Unload all the pieces. This sets the _LastStationDone to 0
METHOD PUBLIC UnloadPieces : BOOL
VAR_INPUT
END_VAR
IF THIS^._LastStationDone <> 0 THEN
    UnloadPieces           := TRUE;
    THIS^._LastStationDone := 0;
    THIS^._ErrorCode       := '';
ELSE
    UnloadPieces := FALSE;
END_IF
END_METHOD

END_FUNCTION_BLOCK

// ---- POUs/20_AUTO/Mover/FB_Station.TcPOU
{attribute 'reflection'}
FUNCTION_BLOCK FB_Station IMPLEMENTS IStation, IObject
VAR_INPUT
END_VAR
VAR_OUTPUT
END_VAR
VAR
    _Position          : REFERENCE TO FB_Position;
    _Process           : REFERENCE TO FB_AUT_ABSTRACT;
    _WaitPosOffset     : LREAL; // offset of the station position, should always be negative
    _iMaxWaitingMovers : INT;   // Maximum of waiting mover in front of the station
    _iGroupNumber      : INT;   // The current group member
    _lrOffset          : LREAL; // offset position of this station for a given recipe
    _bSuperTrackNumber : BYTE;  // target number in superTrack

    _ApproachScenario : ApproachScenario_e := ApproachScenario_e.WaitOnFinishedProcess;

    _iID : INT := 0; // instance ID, is set during FB_Init using the value of _iInstanceCounter 
END_VAR
VAR_STAT
    _iInstanceCounter : INT := 1; // instance counter
END_VAR

PROPERTY ApproachScenario : ApproachScenario_e
GET
ApproachScenario := THIS^._ApproachScenario;
END_GET
SET
THIS^._ApproachScenario := ApproachScenario;
END_SET
END_PROPERTY

METHOD Equals : BOOL
VAR_INPUT
    object : ANY;
END_VAR
Equals := THIS = object.pValue;
END_METHOD

METHOD FB_init : BOOL
VAR_INPUT
    bInitRetains      : BOOL; // if TRUE, the retain variables are initialized (warm start / cold start)
    bInCopyCode       : BOOL; // if TRUE, the instance afterwards gets moved into the copy code (online change)
    Position          : REFERENCE TO FB_Position;
    Process           : REFERENCE TO FB_AUT_ABSTRACT;
    WaitPosOffset     : LREAL;
    ApproachScenario  : ApproachScenario_e;
    iMaxWaitingMovers : INT;
	bSuperTrackNumber : BYTE;
END_VAR
THIS^._iID               := THIS^._iInstanceCounter;
THIS^._iInstanceCounter  := THIS^._iInstanceCounter + 1;
THIS^._Position          REF= Position;
THIS^._Process           REF= Process;
THIS^._WaitPosOffset     := WaitPosOffset;
THIS^._ApproachScenario  := ApproachScenario;
THIS^._iMaxWaitingMovers := iMaxWaitingMovers;
THIS^._bSuperTrackNumber := bSuperTrackNumber;
END_METHOD

PROPERTY GroupNumber : INT
GET
GroupNumber := THIS^._iGroupNumber;
END_GET
SET
THIS^._iGroupNumber := GroupNumber;
END_SET
END_PROPERTY

// the maxuimum number of waiting movers at the front of the station
PROPERTY iMaxWaitingMovers : INT
GET
iMaxWaitingMovers := THIS^._iMaxWaitingMovers;
END_GET
SET
THIS^._iMaxWaitingMovers := iMaxWaitingMovers;
END_SET
END_PROPERTY

PROPERTY PUBLIC Offset : LREAL
GET
Offset := THIS^._lrOffset;
END_GET
SET
THIS^._lrOffset := Offset;
END_SET
END_PROPERTY

PROPERTY Position : REFERENCE TO FB_Position
GET
Position REF=_Position;
END_GET
SET
_Position REF=Position;
END_SET
END_PROPERTY

PROPERTY Process : REFERENCE TO FB_AUT_ABSTRACT
GET
Process REF=_Process;
END_GET
SET
_Process REF= Process;
END_SET
END_PROPERTY

METHOD SetWaitPosOffset : REFERENCE TO FB_Station
VAR_INPUT
	WaitPosOffset : LREAL; // offset position from the given station, must be negative
END_VAR
IF _WaitPosOffset < 0 THEN
    _WaitPosOffset := WaitPos;
END_IF

SetWaitPosOffset REF= THIS^;
END_METHOD

PROPERTY SuperTrackNumber : BYTE
GET
SuperTrackNumber := THIS^._bSuperTrackNumber;
END_GET
END_PROPERTY

METHOD ToString : STRING
VAR_INPUT
END_VAR
VAR_INST
END_VAR
ToString := CONCAT('FB_Station_', TO_STRING(THIS^._iID));
END_METHOD

PROPERTY PUBLIC WaitPos : LREAL
GET
WaitPos := _WaitPosOffset + this^._Position.lrWorkPosition;
END_GET
SET
IF WaitPos < THIS^._Position.lrWorkPosition THEN
    _WaitPosOffset := WaitPos - THIS^._Position.lrWorkPosition;
END_IF
END_SET
END_PROPERTY

END_FUNCTION_BLOCK

// ---- POUs/20_AUTO/Mover/FB_Position.TcPOU
(*
    1D Position class, used to express a given position
	Since the position is in lreal format, you should
	always give a left and a right margin so the isInPosition
	flag will stay stable (beacause we cannot use the = 
	operator on lreal! )
*)
FUNCTION_BLOCK FB_Position IMPLEMENTS IObject
VAR_INPUT
END_VAR
VAR_OUTPUT
END_VAR
VAR
    _lrWorkPosition    : LREAL;      // Work position, use this to give a position
    _lrWorkLeftMargin  : LREAL := 0; // The RELATIVE left position from the work position, need to be POSITIVE
    _lrWorkRightMargin : LREAL := 0; // The RELATIVE right position from the work position, need to be POSITIVE

    _iID : INT := 0; // instance ID, is set during FB_Init using the value of _iInstanceCounter 
END_VAR
VAR_STAT
    _iInstanceCounter : INT := 1; // instance counter
END_VAR

METHOD Equals : BOOL
VAR_INPUT
    object : ANY;
END_VAR
Equals := THIS = object.pValue;
END_METHOD

METHOD FB_init : BOOL
VAR_INPUT
    bInitRetains : BOOL; // if TRUE, the retain variables are initialized (warm start / cold start)
    bInCopyCode  : BOOL; // if TRUE, the instance afterwards gets moved into the copy code (online change)

    lrWorkPosition    : LREAL;      // Work position, use this to give a position
    lrWorkLeftMargin  : LREAL := 0; // The RELATIVE left position from the work position, need to be POSITIVE 
    lrWorkRightMargin : LREAL := 0; // The RELATIVE right position from the work position, need to be POSITIVE
END_VAR
THIS^._iID := THIS^._iInstanceCounter;
THIS^._iInstanceCounter := THIS^._iInstanceCounter +1;
THIS^._lrWorkPosition    := lrWorkPosition;
THIS^._lrWorkLeftMargin  := lrWorkLeftMargin;
THIS^._lrWorkRightMargin := lrWorkRightMargin;
END_METHOD

METHOD isInPos : BOOL
VAR_INPUT
	lrGivenPos : LREAL; // position to test
END_VAR
isInPos := FALSE;

IF ((
    lrGivenPos >= (THIS^._lrWorkPosition - THIS^._lrWorkLeftMargin)) AND
    (lrGivenPos <= (THIS^._lrWorkPosition + THIS^._lrWorkRightMargin)))
    THEN
    isInPos := TRUE;
END_IF
END_METHOD

PROPERTY lrWorkPosition : LREAL
GET
lrWorkPosition := this^._lrWorkPosition;
END_GET
END_PROPERTY

METHOD ToString : STRING
VAR_INPUT
END_VAR
VAR
END_VAR
ToString := CONCAT('FB_Position_', TO_STRING(THIS^._iID));
END_METHOD

END_FUNCTION_BLOCK

// ---- POUs/20_AUTO/ST100/FB_AUT_ABSTRACT.TcPOU
FUNCTION_BLOCK PUBLIC FB_AUT_ABSTRACT IMPLEMENTS IProcessSampleMover
    (****************************************************************************)
    (*	POU_AUT_zxx			Bausteinaufrufe Station	zxx							*)
    (*	Status				ungetestet											*)
    (*  Version:			1.0													*)
    (*	Beschrieb:																*)
    (*																			*)
    (*	Abläufe:			FB_ABLzxxA		Hauptablauf							*)
    (*																			*)
    (*																			*)
    (* 	25.09.2019/Dj															*)
    (****************************************************************************)
    (*	dd.mm.yyyy   KZ    x.y			Beschrieb								*)
    (****************************************************************************)
VAR_INPUT
    (* standart Eingänge *)
    xIN_Init       : BOOL;    // Initialisieren	
    xIN_Quit       : BOOL;    // Fehler quittieren 
    xIN_Start      : BOOL;    // Schrittkette Starten
    xIN_Step       : BOOL;    // Schrittkette Starten/Nachster Schritt
    xIN_ManuCycle  : BOOL;    // Zylus Manuell Starten
    xIN_AlarmAktiv : BOOL;    // Alarm aktiv 
    xIN_DryCycle   : BOOL;    // Fahren ohne Teile 
    enIN_State     : enState; // Status Anlage/Zelle 
    tIN_Timeout    : TIME;    // Timout 
    xIN_On         : BOOL;    // Station eingeschaltet 

    (* spezifische Eingänge *)

END_VAR
VAR_OUTPUT
    (* standart Ausgänge *)
    xOUT_InitDone : BOOL; // fertig initialisiert
    xOUT_Done     : BOOL; // alle Abläufe fertig
    xOUT_Ready    : BOOL; // Station ist bereit (wartet auf Start)
    xOUT_ErrFlag  : BOOL; // Error Flag   
    bOUT_ErrorNum : BYTE; // Error number
    xOUT_Wait     : BOOL; // alle Abläufe warten
    xOUT_AlarmST  : BOOL; // Station hat Alarm

    (* spezifische Ausgänge *)

END_VAR
VAR

    (* Flags *)
    xReset     : BOOL; // Schrittketten zurücksetzen
    xManuCycle : BOOL; // Manueller Zylus aktiv	
    xNextStep  : BOOL; // Nächster Schritt erlaubt	

    xRelease : BOOL := TRUE; // Platzhalter		

    i : INT;

    _iID : INT := 0; // instance ID, is set during FB_Init using the value of _iInstanceCounter 

    _ProcessExecution : ProcessExecution_e := ProcessExecution_e.ExecuteImmediately;

    _Mover             : REFERENCE TO FB_Mover;
    _xMoverShouldLeave : BOOL; // flag to synchronise process and MoverMan, MoverMan needs to call TakeMover() to reset this flag

END_VAR
VAR_STAT
    _iInstanceCounter : INT := 1; // instance counter
END_VAR

METHOD Equals : BOOL
VAR_INPUT
    object : ANY;
END_VAR
Equals := THIS = object.pValue;
END_METHOD

METHOD FB_init : BOOL
VAR_INPUT
	bInitRetains : BOOL; // if TRUE, the retain variables are initialized (warm start / cold start)
	bInCopyCode : BOOL;  // if TRUE, the instance afterwards gets moved into the copy code (online change)
END_VAR
THIS^._iID := THIS^._iInstanceCounter;
THIS^._iInstanceCounter := THIS^._iInstanceCounter +1;
END_METHOD

METHOD GiveMover : IProcessSampleMover
VAR_INPUT
	mover : REFERENCE TO FB_Mover;
END_VAR
IF __ISVALIDREF(THIS^._Mover) THEN
    ASSERT(0); // we already have a mover, this is not permited
ELSIF __ISVALIDREF(mover) THEN
    THIS^._Mover REF= mover;
ELSE
    ASSERT(0); // the given mover is not valid
END_IF
END_METHOD

(* % of completion of the process *)
PROPERTY iCompletionPC : INT
GET
END_GET
END_PROPERTY

(* Process time, expressed in milisecond *)
PROPERTY iProcessTimeMili_1 : DINT
GET
END_GET
SET
END_SET
END_PROPERTY

(* Process time, expressed in milisecond *)
PROPERTY iProcessTimeMili_2 : DINT
GET
END_GET
SET
END_SET
END_PROPERTY

PROPERTY Mover : REFERENCE TO FB_Mover
GET
Mover REF= THIS^._Mover;
END_GET
SET
THIS^._Mover REF= Mover;
END_SET
END_PROPERTY

PROPERTY PUBLIC ProcessExecution : ProcessExecution_e
GET
ProcessExecution := THIS^._ProcessExecution;
END_GET
SET
THIS^._ProcessExecution := ProcessExecution;
END_SET
END_PROPERTY

METHOD TakeMover : IProcessSampleMover
THIS^.Mover REF= 0;
END_METHOD

METHOD ToString : STRING
VAR_INPUT
END_VAR
VAR
END_VAR
ToString := CONCAT('FB_AUT_ABSTRACT_', TO_STRING(THIS^._iID));
END_METHOD

PROPERTY xBusy : BOOL
GET
END_GET
SET
END_SET
END_PROPERTY

PROPERTY xDone : BOOL
GET
END_GET
END_PROPERTY

PROPERTY xMoverPathFree : BOOL
GET
END_GET
END_PROPERTY

PROPERTY xMoverShouldLeave : BOOL
GET
END_GET
END_PROPERTY

END_FUNCTION_BLOCK

// ---- POUs/20_AUTO/Mover/FB_StationMan.TcPOU
FUNCTION_BLOCK FB_StationMan IMPLEMENTS IObject
VAR_INPUT
END_VAR
VAR_OUTPUT
END_VAR
VAR
    // a null terminated array of working station
    _WorkStationList : ARRAY[1..CONST.STATION_NUMBER] OF POINTER TO FB_Station;
    _PieceHolder     : REFERENCE TO FB_PieceHolder;

    _GroupList : ARRAY[1..CONST.MAX_GROUP] OF FB_Group;

    _iID : INT := 0; // instance ID, is set during FB_Init using the value of _iInstanceCounter 
END_VAR
VAR_STAT
    _iInstanceCounter : INT := 1; // instance counter
END_VAR

METHOD Equals : BOOL
VAR_INPUT
    object : ANY;
END_VAR
Equals := THIS = object.pValue;
END_METHOD

METHOD FB_init : BOOL
VAR_INPUT
    bInitRetains : BOOL; // if TRUE, the retain variables are initialized (warm start / cold start)
    bInCopyCode  : BOOL; // if TRUE, the instance afterwards gets moved into the copy code (online change)

    // The full station list of the application
    StationList : POINTER TO ARRAY[1..CONST.STATION_NUMBER] OF FB_Station;
    // Used to determine which station is used
    SelStationList : POINTER TO ARRAY[1..CONST.STATION_NUMBER] OF INT;
    PieceHolder    : REFERENCE TO FB_PieceHolder;

END_VAR
VAR
    i                 : INT;
    selStationCounter : INT := 1;
END_VAR
THIS^._iID              := THIS^._iInstanceCounter;
THIS^._iInstanceCounter := THIS^._iInstanceCounter + 1;

FOR i := 1 TO const.STATION_NUMBER BY 1 DO
    IF SelStationList^[i] >= 0 THEN
        THIS^._WorkStationList[selStationCounter] := ADR(StationList^[i]);

        selStationCounter := selStationCounter + 1;
    END_IF
END_FOR

_PieceHolder REF= PieceHolder;
THIS^.SetGroupMembers(StationList, SelStationList);
END_METHOD

// Return the closest station using the station position 
// First we search if we are in range with our set of station
// then, if no station are in our range, we give the nearest next
// station
METHOD PRIVATE FindCloserStationIndex : INT
VAR_INPUT
    CurrentPosition : LREAL;
END_VAR
VAR
    i : INT;
END_VAR
FindCloserStationIndex := -1;

// First we check if we are not in range of a station from our set
FOR i := 1 TO CONST.STATION_NUMBER BY 1 DO
    IF 0 <> THIS^._WorkStationList[i] THEN
        IF THIS^._WorkStationList[i]^.Position.isInPos(CurrentPosition) THEN
            FindCloserStationIndex := i;
            RETURN;
        END_IF
    END_IF
END_FOR

// Then, if no station are in the range, we give the most nearest station, if possible
FOR i := 1 TO CONST.STATION_NUMBER BY 1 DO
    IF 0 <> THIS^._WorkStationList[i] THEN
        IF __ISVALIDREF(THIS^._WorkStationList[i]^.Position) AND
           THIS^._WorkStationList[i]^.Position.lrWorkPosition > CurrentPosition THEN
            FindCloserStationIndex := i;
            EXIT;
        END_IF
    END_IF
END_FOR
END_METHOD

// Return the next station to visit
METHOD GetNextStation : REFERENCE TO FB_Station
VAR_INPUT
    CurrentStation : REFERENCE TO FB_Station;
END_VAR
VAR
    CurrStationIndex : INT;
END_VAR
GetNextStation   REF= CurrentStation;
CurrStationIndex := THIS^.GetStationIndex(CurrentStation);

IF CurrStationIndex > 0 THEN

    IF CurrentStation.GroupNumber > 0 THEN
		// We search for a station which is not from the same group
        WHILE GetNextStation.GroupNumber = CurrentStation.GroupNumber DO
            CurrStationIndex := THIS^.GetNextStationIndex(CurrStationIndex);
            GetNextStation   REF= THIS^._WorkStationList[CurrStationIndex]^;
        END_WHILE
    ELSE
        CurrStationIndex := THIS^.GetNextStationIndex(CurrStationIndex);
        GetNextStation   REF= THIS^._WorkStationList[CurrStationIndex]^;
    END_IF

    // We take a look of the group member and then set the corresponding station
    IF GetNextStation.GroupNumber > 0 THEN
        GetNextStation REF= THIS^._GroupList[GetNextStation.GroupNumber].GetNextStation();
    END_IF

    // when the current is not on the list, we try to move to the nearest
    // but only on the positive direction
ELSE
    CurrStationIndex := THIS^.FindCloserStationIndex(CurrentStation.Position.lrWorkPosition);

    IF CurrStationIndex > 0 THEN
        GetNextStation REF= THIS^._WorkStationList[CurrStationIndex]^;

    ELSE
        GetNextStation REF= THIS^._WorkStationList[1]^;

    END_IF
END_IF
END_METHOD

// Return the next station index in the ring buffer of station
METHOD PRIVATE GetNextStationIndex : INT
VAR_INPUT
	CurrStationIndex : INT;
END_VAR
IF CurrStationIndex >= CONST.STATION_NUMBER THEN
    GetNextStationIndex := 1;

ELSIF THIS^._WorkStationList[CurrStationIndex + 1] = 0 THEN
    GetNextStationIndex := 1;

ELSE
    GetNextStationIndex := CurrStationIndex + 1;
END_IF
END_METHOD

// Get the next station with a valid process. If nothing is found, we 
// simply return to the first station (this should be never the case
// since your machine will be useless...)
METHOD GetNextStationWithProcess : REFERENCE TO FB_Station
VAR_INPUT
    CurrentStation : REFERENCE TO FB_Station;
END_VAR
VAR
    // search station with process algorithme
    iSearchNext        : INT; // incremtal variable used to search in a set of next station
    iTempSearchStation : INT; // incremtal variable used to search in a set of next station
    tempStation        : REFERENCE TO FB_Station;
END_VAR
// If nothing found, we return to the first station
GetNextStationWithProcess REF= THIS^._WorkStationList[1]^;

IF __ISVALIDREF(CurrentStation) THEN
    iSearchNext := 1;

    WHILE iSearchNext < CONST.STATION_NUMBER DO
        tempStation REF= THIS^.GetNextStation(CurrentStation);

        IF __ISVALIDREF(tempStation) AND_THEN __ISVALIDREF(tempStation.Process) THEN
            GetNextStationWithProcess REF= tempStation;
            EXIT;
        END_IF

        iSearchNext := iSearchNext + 1;

    END_WHILE
END_IF
END_METHOD

METHOD GetStartStation : POINTER TO FB_Station
VAR_INPUT
    CurrentPosition : LREAL;
END_VAR
VAR
    CurrStationIndex : INT;
END_VAR
//GetStartStation := THIS^._WorkStationList[1];
CurrStationIndex := THIS^.FindCloserStationIndex(CurrentPosition);

IF CurrStationIndex > 0 THEN
    GetStartStation := THIS^._WorkStationList[CurrStationIndex];

ELSE
    GetStartStation := THIS^._WorkStationList[1];

END_IF
END_METHOD

// return the index of a given station, If the index is -1, no station where found
METHOD PRIVATE GetStationIndex : INT
VAR_INPUT
    Station : REFERENCE TO FB_Station;
END_VAR
VAR
    i : INT;
END_VAR
GetStationIndex := -1;

FOR i := 1 TO CONST.STATION_NUMBER BY 1 DO
    IF Station.Equals(THIS^._WorkStationList[i]^) THEN
        GetStationIndex := i;
        EXIT;
    END_IF
END_FOR
END_METHOD

PROPERTY PieceHolder : REFERENCE TO FB_PieceHolder
GET
PieceHolder REF= _PieceHolder;
END_GET
SET
_PieceHolder REF= PieceHolder;
END_SET
END_PROPERTY

METHOD SetGroupMembers : REFERENCE TO FB_Group
VAR_INPUT
    // The full station list of the application
    StationList : POINTER TO ARRAY[1..CONST.STATION_NUMBER] OF FB_Station;
    SelStationList : POINTER TO ARRAY[1..CONST.STATION_NUMBER] OF INT;
END_VAR
VAR
    i : INT;
END_VAR
FOR i := 1 TO CONST.STATION_NUMBER BY 1 DO
    IF SelStationList^[i] > 0 AND SelStationList^[i] <= CONST.MAX_GROUP THEN
        THIS^._GroupList[SelStationList^[i]].AddStation(StationList^[i]);
		StationList^[i].GroupNumber := SelStationList^[i];
    END_IF
END_FOR
END_METHOD

METHOD ToString : STRING
VAR_INPUT
END_VAR
VAR
END_VAR
ToString := CONCAT('FB_StationMan_', TO_STRING(THIS^._iID));
END_METHOD

END_FUNCTION_BLOCK

// ---- POUs/20_AUTO/Mover/FB_Group.TcPOU
// Create station group and manage shuttle behaviour 
FUNCTION_BLOCK FB_Group IMPLEMENTS IObject
VAR_INPUT
END_VAR
VAR_OUTPUT
END_VAR
VAR
    _GroupNumber : INT; // group number

    _StationList : ARRAY[1..CONST.MAX_STATION_PER_GROUP] OF POINTER TO FB_Station; // Array of member station member

    _LastVisitedIndex : INT; // Last visited station index
    _MaxStationList   : INT; // The current maximum of station in this group. 0 means no station are present
	
	_iID : INT := 0; // instance ID, is set during FB_Init using the value of _iInstanceCounter 
END_VAR
VAR_STAT
	_iInstanceCounter : INT; // instance counter
END_VAR

METHOD AddStation : REFERENCE TO FB_Group
VAR_INPUT
    station : REFERENCE TO FB_Station;
END_VAR
IF THIS^._MaxStationList < CONST.MAX_STATION_PER_GROUP THEN
    THIS^._MaxStationList                     := THIS^._MaxStationList + 1;
    THIS^._StationList[THIS^._MaxStationList] := ADR(station);
ELSE
    ASSERT(0);
END_IF
END_METHOD

METHOD Equals : BOOL
VAR_INPUT
    object : ANY;
END_VAR
Equals := THIS = object.pValue;
END_METHOD

METHOD FB_init : BOOL
VAR_INPUT
    bInitRetains : BOOL; // if TRUE, the retain variables are initialized (warm start / cold start)
    bInCopyCode  : BOOL; // if TRUE, the instance afterwards gets moved into the copy code (online change)
END_VAR
THIS^._iInstanceCounter := THIS^._iInstanceCounter + 1;
THIS^._iID              := THIS^._iInstanceCounter;

THIS^._MaxStationList   := 0;
THIS^._LastVisitedIndex := 1; // the last station is set to the first

IF THIS^._iID <= CONST.MAX_GROUP THEN
    THIS^._GroupNumber := THIS^._iID;
ELSE
    ASSERT(0);
END_IF
END_METHOD

// The next station is always the one before the last visited
METHOD GetNextStation : REFERENCE TO FB_Station
VAR_INPUT
END_VAR
(* Note about this algorithme :
 * The goal of this algorithm is to divide equaly the use of each station
 * so the wear of station is the same. Other algorithm can be implemented 
 * if needed.
*)
IF THIS^._LastVisitedIndex <= 1 THEN
    THIS^._LastVisitedIndex := THIS^._MaxStationList;
ELSE
    THIS^._LastVisitedIndex := THIS^._LastVisitedIndex - 1;
END_IF

GetNextStation REF= THIS^._StationList[THIS^._LastVisitedIndex]^;
END_METHOD

PROPERTY GroupNumber : INT
GET
GroupNumber := this^._GroupNumber;
END_GET
END_PROPERTY

METHOD ToString : STRING
VAR_INPUT
END_VAR
ToString := CONCAT('FB_Station_', TO_STRING(THIS^._iID));
END_METHOD

END_FUNCTION_BLOCK

// ---- POUs/20_AUTO/_20_AUTO.TcPOU
PROGRAM
    _20_AUTO
VAR_INPUT
    xIN_Quit   : BOOL;    //Quittieren
    enIN_State : enState; //Status der Maschine 
    recipe     : REFERENCE TO Recipe_21_101_t;
END_VAR
VAR_OUTPUT
END_VAR
VAR
    recipeHMI       : REFERENCE TO Recipe_21_101_t;                // recipe values shown on the HMI
    iRecipeCopyDest : RecipeType_e := RecipeType_e._max  ; // selected recipe to copy to
	fb_axis130_01Z : FB_AxisLIN_V1_1;
END_VAR

//Alarm Allgemein
//POU_ERR_000(xIN_QUIT:=xIN_Quit , pstrArIN_ALARM:=ADR(HMI.strArALARM[1]));
//POU_MSG_000(xIN_QUIT:=xIN_Quit , pstrArIN_ALARM:=ADR(HMI.strArMSG[1]));

recipeHMI REF= PERS.recipeList[PERS.iRecipeCurrent];
recipe    REF= PERS.recipeList[PERS.iRecipeCurrent];

PERS.iRecipeCurrent := PERS.eRecipeCurrent;

IF HMI.btCopyRecipe.rtrig THEN
    PERS.recipeList[iRecipeCopyDest] := PERS.recipeList[PERS.iRecipeCurrent];
    // reset the position of iRecipeCopyDest to tell the user the saving is done
    iRecipeCopyDest := RecipeType_e._max;
END_IF

IF HMI.btSetDefault.rtrig THEN
    _21_CopyDefaultRecipe();
END_IF

IF HMI.btCopyAxisCfg.rtrig THEN
    PERS.recipeList[PERS.iRecipeCurrent].linearAxis[HMI.iSelectAxisCopy] :=
        PERS.recipeList[PERS.iRecipeCurrent].linearAxis[HMI.iSelectAxis];

    // reset the position of iRecipeCopyDest to tell the user the saving is done
    HMI.iSelectAxisCopy := TO_INT(LinearAxis_e._max);
END_IF

IF HMI.btCopyCylinderCfg.rtrig THEN
    PERS.recipeList[PERS.iRecipeCurrent].cylinder2Pos[HMI.iSelectCylinderCopy] :=
        PERS.recipeList[PERS.iRecipeCurrent].cylinder2Pos[HMI.iSelectCylinder];

    // reset the position of iRecipeCopyDest to tell the user the saving is done
    HMI.iSelectCylinderCopy := TO_INT(StationList_e._max);
END_IF

//Station01

SIMU.iCompletionHMI[StationList_e.ST105 + 1] := GVL.st105_aut.iCompletionPC;
GVL.st105_aut.iProcessTimeMili_1             := PERS.iStationTimeDef1[StationList_e.ST105 + 1];
GVL.st105_aut.iProcessTimeMili_2             := PERS.iStationTimeDef2[StationList_e.ST105 + 1];

GVL.st105_aut(xIN_Init       := HMI.enState = enState.StateINIT,
              xIN_Start      := HMI.btArMain[9].press,
              xIN_Step       := HMI.btArMain[1].rtrig,
              xIN_ManuCycle  := HMI.enState = StateMANU,
              xIN_Quit       := xIN_Quit,
              xIN_AlarmAktiv := HMI.xAlarm,
              xIN_DryCycle   := FALSE,
              enIN_State     := enIN_State,
              tIN_Timeout    := T#10S,
              xIN_On         := TRUE);

SIMU.iCompletionHMI[StationList_e.ST110 + 1] := GVL.st110_aut.iCompletionPC;
GVL.st110_aut.iProcessTimeMili_1             := PERS.iStationTimeDef1[StationList_e.ST110 + 1];
GVL.st110_aut.iProcessTimeMili_2             := PERS.iStationTimeDef2[StationList_e.ST110 + 1];
GVL.st110_aut(xIN_Init       := HMI.enState = enState.StateINIT,
              xIN_Start      := HMI.btArMain[9].press,
              xIN_Step       := HMI.btArMain[1].rtrig,
              xIN_ManuCycle  := HMI.enState = StateMANU,
              xIN_Quit       := xIN_Quit,
              xIN_AlarmAktiv := HMI.xAlarm,
              xIN_DryCycle   := FALSE,
              enIN_State     := enIN_State,
              tIN_Timeout    := T#10S,
              xIN_On         := TRUE);

SIMU.iCompletionHMI[StationList_e.ST115 + 1] := GVL.st115_aut.iCompletionPC;
GVL.st115_aut.iProcessTimeMili_1             := PERS.iStationTimeDef1[StationList_e.ST115 + 1];
GVL.st115_aut.iProcessTimeMili_2             := PERS.iStationTimeDef2[StationList_e.ST115 + 1];
GVL.st115_aut(xIN_Init       := HMI.enState = enState.StateINIT,
              xIN_Start      := HMI.btArMain[9].press,
              xIN_Step       := HMI.btArMain[1].rtrig,
              xIN_ManuCycle  := HMI.enState = StateMANU,
              xIN_Quit       := xIN_Quit,
              xIN_AlarmAktiv := HMI.xAlarm,
              xIN_DryCycle   := FALSE,
              enIN_State     := enIN_State,
              tIN_Timeout    := T#10S,
              xIN_On         := TRUE);

SIMU.iCompletionHMI[StationList_e.ST120 + 1] := GVL.st120_aut.iCompletionPC;
GVL.st120_aut.iProcessTimeMili_1             := PERS.iStationTimeDef1[StationList_e.ST120 + 1];
GVL.st120_aut.iProcessTimeMili_2             := PERS.iStationTimeDef2[StationList_e.ST120 + 1];
GVL.st120_aut(xIN_Init       := HMI.enState = enState.StateINIT,
              xIN_Start      := HMI.btArMain[9].press,
              xIN_Step       := HMI.btArMain[1].rtrig,
              xIN_ManuCycle  := HMI.enState = StateMANU,
              xIN_Quit       := xIN_Quit,
              xIN_AlarmAktiv := HMI.xAlarm,
              xIN_DryCycle   := FALSE,
              enIN_State     := enIN_State,
              tIN_Timeout    := T#10S,
              xIN_On         := TRUE);

SIMU.iCompletionHMI[StationList_e.ST125 + 1] := GVL.st125_aut.iCompletionPC;
GVL.st125_aut.iProcessTimeMili_1             := PERS.iStationTimeDef1[StationList_e.ST125 + 1];
GVL.st125_aut.iProcessTimeMili_2             := PERS.iStationTimeDef2[StationList_e.ST125 + 1];
GVL.st125_aut(xIN_Init       := HMI.enState = enState.StateINIT,
              xIN_Start      := HMI.btArMain[9].press,
              xIN_Step       := HMI.btArMain[1].rtrig,
              xIN_ManuCycle  := HMI.enState = StateMANU,
              xIN_Quit       := xIN_Quit,
              xIN_AlarmAktiv := HMI.xAlarm,
              xIN_DryCycle   := FALSE,
              enIN_State     := enIN_State,
              tIN_Timeout    := T#10S,
              xIN_On         := TRUE);

SIMU.iCompletionHMI[StationList_e.ST128 + 1] := GVL.st125_aut.iCompletionPC;
GVL.st128_aut.iProcessTimeMili_1             := PERS.iStationTimeDef1[StationList_e.ST128 + 1];
GVL.st128_aut.iProcessTimeMili_2             := PERS.iStationTimeDef2[StationList_e.ST128 + 1];
GVL.st128_aut(xIN_Init       := HMI.enState = enState.StateINIT,
              xIN_Start      := HMI.btArMain[9].press,
              xIN_Step       := HMI.btArMain[1].rtrig,
              xIN_ManuCycle  := HMI.enState = StateMANU,
              xIN_Quit       := xIN_Quit,
              xIN_AlarmAktiv := HMI.xAlarm,
              xIN_DryCycle   := FALSE,
              enIN_State     := enIN_State,
              tIN_Timeout    := T#10S,
              xIN_On         := TRUE);

SIMU.iCompletionHMI[StationList_e.ST130 + 1] := GVL.st130_aut.iCompletionPC;
GVL.st130_aut.iProcessTimeMili_1             := PERS.iStationTimeDef1[StationList_e.ST130 + 1];
GVL.st130_aut.iProcessTimeMili_2             := PERS.iStationTimeDef2[StationList_e.ST130 + 1];
GVL.st130_aut(xIN_Init       := HMI.enState = enState.StateINIT,
              xIN_Start      := HMI.btArMain[9].press,
              xIN_Step       := HMI.btArMain[1].rtrig,
              xIN_ManuCycle  := HMI.enState = StateMANU,
              xIN_Quit       := xIN_Quit,
              xIN_AlarmAktiv := HMI.xAlarm,
              xIN_DryCycle   := FALSE,
              enIN_State     := enIN_State,
              tIN_Timeout    := T#10S,
              xIN_On         := TRUE);

SIMU.iCompletionHMI[StationList_e.ST135 + 1] := GVL.st135_aut.iCompletionPC;
GVL.st135_aut.iProcessTimeMili_1             := PERS.iStationTimeDef1[StationList_e.ST135 + 1];
GVL.st135_aut.iProcessTimeMili_2             := PERS.iStationTimeDef2[StationList_e.ST135 + 1];
GVL.st135_aut(xIN_Init       := HMI.enState = enState.StateINIT,
              xIN_Start      := HMI.btArMain[9].press,
              xIN_Step       := HMI.btArMain[1].rtrig,
              xIN_ManuCycle  := HMI.enState = StateMANU,
              xIN_Quit       := xIN_Quit,
              xIN_AlarmAktiv := HMI.xAlarm,
              xIN_DryCycle   := FALSE,
              enIN_State     := enIN_State,
              tIN_Timeout    := T#10S,
              xIN_On         := TRUE);

SIMU.iCompletionHMI[StationList_e.ST140 + 1] := GVL.st140_aut.iCompletionPC;
GVL.st140_aut.iProcessTimeMili_1             := PERS.iStationTimeDef1[StationList_e.ST140 + 1];
GVL.st140_aut.iProcessTimeMili_2             := PERS.iStationTimeDef2[StationList_e.ST140 + 1];
GVL.st140_aut(xIN_Init       := HMI.enState = enState.StateINIT,
              xIN_Start      := HMI.btArMain[9].press,
              xIN_Step       := HMI.btArMain[1].rtrig,
              xIN_ManuCycle  := HMI.enState = StateMANU,
              xIN_Quit       := xIN_Quit,
              xIN_AlarmAktiv := HMI.xAlarm,
              xIN_DryCycle   := FALSE,
              enIN_State     := enIN_State,
              tIN_Timeout    := T#10S,
              xIN_On         := TRUE);

SIMU.iCompletionHMI[StationList_e.ST145 + 1] := GVL.st145_aut.iCompletionPC;
GVL.st145_aut.iProcessTimeMili_1             := PERS.iStationTimeDef1[StationList_e.ST145 + 1];
GVL.st145_aut.iProcessTimeMili_2             := PERS.iStationTimeDef2[StationList_e.ST145 + 1];
GVL.st145_aut(xIN_Init       := HMI.enState = enState.StateINIT,
              xIN_Start      := HMI.btArMain[9].press,
              xIN_Step       := HMI.btArMain[1].rtrig,
              xIN_ManuCycle  := HMI.enState = StateMANU,
              xIN_Quit       := xIN_Quit,
              xIN_AlarmAktiv := HMI.xAlarm,
              xIN_DryCycle   := FALSE,
              enIN_State     := enIN_State,
              tIN_Timeout    := T#10S,
              xIN_On         := TRUE);

SIMU.iCompletionHMI[StationList_e.ST150 + 1] := GVL.st150_aut.iCompletionPC;
GVL.st150_aut.iProcessTimeMili_1             := PERS.iStationTimeDef1[StationList_e.ST150 + 1];
GVL.st150_aut.iProcessTimeMili_2             := PERS.iStationTimeDef2[StationList_e.ST150 + 1];
GVL.st150_aut(xIN_Init       := HMI.enState = enState.StateINIT,
              xIN_Start      := HMI.btArMain[9].press,
              xIN_Step       := HMI.btArMain[1].rtrig,
              xIN_ManuCycle  := HMI.enState = StateMANU,
              xIN_Quit       := xIN_Quit,
              xIN_AlarmAktiv := HMI.xAlarm,
              xIN_DryCycle   := FALSE,
              enIN_State     := enIN_State,
              tIN_Timeout    := T#10S,
              xIN_On         := TRUE);

SIMU.iCompletionHMI[StationList_e.ST155 + 1] := GVL.st155_aut.iCompletionPC;
GVL.st155_aut.iProcessTimeMili_1             := PERS.iStationTimeDef1[StationList_e.ST155 + 1];
GVL.st155_aut.iProcessTimeMili_2             := PERS.iStationTimeDef2[StationList_e.ST155 + 1];
GVL.st155_aut(xIN_Init       := HMI.enState = enState.StateINIT,
              xIN_Start      := HMI.btArMain[9].press,
              xIN_Step       := HMI.btArMain[1].rtrig,
              xIN_ManuCycle  := HMI.enState = StateMANU,
              xIN_Quit       := xIN_Quit,
              xIN_AlarmAktiv := HMI.xAlarm,
              xIN_DryCycle   := FALSE,
              enIN_State     := enIN_State,
              tIN_Timeout    := T#10S,
              xIN_On         := TRUE);

SIMU.iCompletionHMI[StationList_e.ST160 + 1] := GVL.st160_aut.iCompletionPC;
GVL.st160_aut.iProcessTimeMili_1             := PERS.iStationTimeDef1[StationList_e.ST160 + 1];
GVL.st160_aut.iProcessTimeMili_2             := PERS.iStationTimeDef2[StationList_e.ST160 + 1];
GVL.st160_aut(xIN_Init       := HMI.enState = enState.StateINIT,
              xIN_Start      := HMI.btArMain[9].press,
              xIN_Step       := HMI.btArMain[1].rtrig,
              xIN_ManuCycle  := HMI.enState = StateMANU,
              xIN_Quit       := xIN_Quit,
              xIN_AlarmAktiv := HMI.xAlarm,
              xIN_DryCycle   := FALSE,
              enIN_State     := enIN_State,
              tIN_Timeout    := T#10S,
              xIN_On         := TRUE);

SIMU.iCompletionHMI[StationList_e.ST165 + 1] := GVL.st165_aut.iCompletionPC;
GVL.st165_aut.iProcessTimeMili_1             := PERS.iStationTimeDef1[StationList_e.ST165 + 1];
GVL.st165_aut.iProcessTimeMili_2             := PERS.iStationTimeDef2[StationList_e.ST165 + 1];
GVL.st165_aut(xIN_Init       := HMI.enState = enState.StateINIT,
              xIN_Start      := HMI.btArMain[9].press,
              xIN_Step       := HMI.btArMain[1].rtrig,
              xIN_ManuCycle  := HMI.enState = StateMANU,
              xIN_Quit       := xIN_Quit,
              xIN_AlarmAktiv := HMI.xAlarm,
              xIN_DryCycle   := FALSE,
              enIN_State     := enIN_State,
              tIN_Timeout    := T#10S,
              xIN_On         := TRUE);

SIMU.iCompletionHMI[StationList_e.ST170 + 1] := GVL.st170_aut.iCompletionPC;
GVL.st170_aut.iProcessTimeMili_1             := PERS.iStationTimeDef1[StationList_e.ST170 + 1];
GVL.st170_aut.iProcessTimeMili_2             := PERS.iStationTimeDef2[StationList_e.ST170 + 1];
GVL.st170_aut(xIN_Init       := HMI.enState = enState.StateINIT,
              xIN_Start      := HMI.btArMain[9].press,
              xIN_Step       := HMI.btArMain[1].rtrig,
              xIN_ManuCycle  := HMI.enState = StateMANU,
              xIN_Quit       := xIN_Quit,
              xIN_AlarmAktiv := HMI.xAlarm,
              xIN_DryCycle   := FALSE,
              enIN_State     := enIN_State,
              tIN_Timeout    := T#10S,
              xIN_On         := TRUE);

SIMU.iCompletionHMI[StationList_e.ST175 + 2] := GVL.st175_aut.iCompletionPC;
GVL.st175_aut.iProcessTimeMili_1             := PERS.iStationTimeDef1[StationList_e.ST175 + 2];
GVL.st175_aut.iProcessTimeMili_2             := PERS.iStationTimeDef2[StationList_e.ST175 + 2];
GVL.st175_aut(xIN_Init       := HMI.enState = enState.StateINIT,
              xIN_Start      := HMI.btArMain[9].press,
              xIN_Step       := HMI.btArMain[1].rtrig,
              xIN_ManuCycle  := HMI.enState = StateMANU,
              xIN_Quit       := xIN_Quit,
              xIN_AlarmAktiv := HMI.xAlarm,
              xIN_DryCycle   := FALSE,
              enIN_State     := enIN_State,
              tIN_Timeout    := T#10S,
              xIN_On         := TRUE);

SIMU.iCompletionHMI[StationList_e.ST176 + 2] := GVL.st176_aut.iCompletionPC;
GVL.st176_aut.iProcessTimeMili_1             := PERS.iStationTimeDef1[StationList_e.ST176 + 2];
GVL.st176_aut.iProcessTimeMili_2             := PERS.iStationTimeDef2[StationList_e.ST176 + 2];
GVL.st176_aut(xIN_Init       := HMI.enState = enState.StateINIT,
              xIN_Start      := HMI.btArMain[9].press,
              xIN_Step       := HMI.btArMain[1].rtrig,
              xIN_ManuCycle  := HMI.enState = StateMANU,
              xIN_Quit       := xIN_Quit,
              xIN_AlarmAktiv := HMI.xAlarm,
              xIN_DryCycle   := FALSE,
              enIN_State     := enIN_State,
              tIN_Timeout    := T#10S,
              xIN_On         := TRUE);

SIMU.iCompletionHMI[StationList_e.ST180 + 2] := GVL.st180_aut.iCompletionPC;
GVL.st180_aut.iProcessTimeMili_1             := PERS.iStationTimeDef1[StationList_e.ST180 + 2];
GVL.st180_aut.iProcessTimeMili_2             := PERS.iStationTimeDef2[StationList_e.ST180 + 2];
GVL.st180_aut(xIN_Init       := HMI.enState = enState.StateINIT,
              xIN_Start      := HMI.btArMain[9].press,
              xIN_Step       := HMI.btArMain[1].rtrig,
              xIN_ManuCycle  := HMI.enState = StateMANU,
              xIN_Quit       := xIN_Quit,
              xIN_AlarmAktiv := HMI.xAlarm,
              xIN_DryCycle   := FALSE,
              enIN_State     := enIN_State,
              tIN_Timeout    := T#10S,
              xIN_On         := TRUE);

SIMU.iCompletionHMI[StationList_e.ST185 + 2] := GVL.st185_aut.iCompletionPC;
GVL.st185_aut.iProcessTimeMili_1             := PERS.iStationTimeDef1[StationList_e.ST185 + 2];
GVL.st185_aut.iProcessTimeMili_2             := PERS.iStationTimeDef2[StationList_e.ST185 + 2];
GVL.st185_aut(xIN_Init       := HMI.enState = enState.StateINIT,
              xIN_Start      := HMI.btArMain[9].press,
              xIN_Step       := HMI.btArMain[1].rtrig,
              xIN_ManuCycle  := HMI.enState = StateMANU,
              xIN_Quit       := xIN_Quit,
              xIN_AlarmAktiv := HMI.xAlarm,
              xIN_DryCycle   := FALSE,
              enIN_State     := enIN_State,
              tIN_Timeout    := T#10S,
              xIN_On         := TRUE);

END_PROGRAM

// ---- POUs/20_AUTO/_21_CopyDefaultRecipe.TcPOU
FUNCTION _21_CopyDefaultRecipe : BOOL
VAR_INPUT
END_VAR
VAR
    i  : INT;
    ii : INT;
END_VAR


FOR i := 0 TO TO_INT(LinearAxis_e._max) - 1 BY 1 DO
    PERS.recipeList[0].linearAxis[i].defProfile.lrVelocity := 100;
    PERS.recipeList[0].linearAxis[i].defProfile.lrAccel    := 5000;
    PERS.recipeList[0].linearAxis[i].defProfile.lrDecel    := 5000;
    PERS.recipeList[0].linearAxis[i].defProfile.lrJerk     := 500000;
END_FOR

// ST110
PERS.recipeList[0].linearAxis[LinearAxis_e.ST110_01Y].movesList[0].lrPosition := 10;
PERS.recipeList[0].linearAxis[LinearAxis_e.ST110_01Y].movesList[1].lrPosition := 100;

PERS.recipeList[0].linearAxis[LinearAxis_e.ST110_02Z].movesList[0].lrPosition := 10;
PERS.recipeList[0].linearAxis[LinearAxis_e.ST110_02Z].movesList[1].lrPosition := 50;
PERS.recipeList[0].linearAxis[LinearAxis_e.ST110_02Z].movesList[2].lrPosition := 2;
PERS.recipeList[0].linearAxis[LinearAxis_e.ST110_02Z].movesList[3].lrPosition := 50;
PERS.recipeList[0].linearAxis[LinearAxis_e.ST110_02Z].movesList[4].lrPosition := 80;

PERS.recipeList[0].linearAxis[LinearAxis_e.ST110_03Z].movesList[0].lrPosition := 10;
PERS.recipeList[0].linearAxis[LinearAxis_e.ST110_03Z].movesList[1].lrPosition := 50;
PERS.recipeList[0].linearAxis[LinearAxis_e.ST110_03Z].movesList[2].lrPosition := 2;
PERS.recipeList[0].linearAxis[LinearAxis_e.ST110_03Z].movesList[3].lrPosition := 50;
PERS.recipeList[0].linearAxis[LinearAxis_e.ST110_03Z].movesList[4].lrPosition := 80;

PERS.recipeList[0].linearAxis[LinearAxis_e.ST110_04Z].movesList[0].lrPosition := 10;
PERS.recipeList[0].linearAxis[LinearAxis_e.ST110_04Z].movesList[1].lrPosition := 50;

// ST115
PERS.recipeList[0].linearAxis[LinearAxis_e.ST115_01Y].movesList[0].lrPosition := 10;
PERS.recipeList[0].linearAxis[LinearAxis_e.ST115_01Y].movesList[1].lrPosition := 100;

PERS.recipeList[0].linearAxis[LinearAxis_e.ST115_02Z].movesList[0].lrPosition := 10;
PERS.recipeList[0].linearAxis[LinearAxis_e.ST115_02Z].movesList[1].lrPosition := 50;
PERS.recipeList[0].linearAxis[LinearAxis_e.ST115_02Z].movesList[2].lrPosition := 2;
PERS.recipeList[0].linearAxis[LinearAxis_e.ST115_02Z].movesList[3].lrPosition := 50;
PERS.recipeList[0].linearAxis[LinearAxis_e.ST115_02Z].movesList[4].lrPosition := 80;

PERS.recipeList[0].linearAxis[LinearAxis_e.ST115_03Z].movesList[0].lrPosition := 10;
PERS.recipeList[0].linearAxis[LinearAxis_e.ST115_03Z].movesList[1].lrPosition := 50;
PERS.recipeList[0].linearAxis[LinearAxis_e.ST115_03Z].movesList[2].lrPosition := 2;
PERS.recipeList[0].linearAxis[LinearAxis_e.ST115_03Z].movesList[3].lrPosition := 50;
PERS.recipeList[0].linearAxis[LinearAxis_e.ST115_03Z].movesList[4].lrPosition := 80;

PERS.recipeList[0].linearAxis[LinearAxis_e.ST115_04Z].movesList[0].lrPosition := 10;
PERS.recipeList[0].linearAxis[LinearAxis_e.ST115_04Z].movesList[1].lrPosition := 50;

// ST120
PERS.recipeList[0].linearAxis[LinearAxis_e.ST120_01Y].movesList[0].lrPosition := 10;
PERS.recipeList[0].linearAxis[LinearAxis_e.ST120_01Y].movesList[1].lrPosition := 100;

PERS.recipeList[0].linearAxis[LinearAxis_e.ST120_02Z].movesList[0].lrPosition := 10;
PERS.recipeList[0].linearAxis[LinearAxis_e.ST120_02Z].movesList[1].lrPosition := 50;
PERS.recipeList[0].linearAxis[LinearAxis_e.ST120_02Z].movesList[2].lrPosition := 2;
PERS.recipeList[0].linearAxis[LinearAxis_e.ST120_02Z].movesList[3].lrPosition := 50;
PERS.recipeList[0].linearAxis[LinearAxis_e.ST120_02Z].movesList[4].lrPosition := 80;

// ST125
PERS.recipeList[0].linearAxis[LinearAxis_e.ST125_01Y].movesList[0].lrPosition := 10;
PERS.recipeList[0].linearAxis[LinearAxis_e.ST125_01Y].movesList[1].lrPosition := 100;

PERS.recipeList[0].linearAxis[LinearAxis_e.ST125_02Z].movesList[0].lrPosition := 10;
PERS.recipeList[0].linearAxis[LinearAxis_e.ST125_02Z].movesList[1].lrPosition := 50;
PERS.recipeList[0].linearAxis[LinearAxis_e.ST125_02Z].movesList[2].lrPosition := 2;
PERS.recipeList[0].linearAxis[LinearAxis_e.ST125_02Z].movesList[3].lrPosition := 50;
PERS.recipeList[0].linearAxis[LinearAxis_e.ST125_02Z].movesList[4].lrPosition := 80;
PERS.recipeList[0].linearAxis[LinearAxis_e.ST125_02Z].movesList[5].lrPosition := 50;

// ST130
PERS.recipeList[0].linearAxis[LinearAxis_e.ST130_01Z].movesList[0].lrPosition := 10;
PERS.recipeList[0].linearAxis[LinearAxis_e.ST130_01Z].movesList[1].lrPosition := 260;

PERS.recipeList[0].linearAxis[LinearAxis_e.ST130_10Z].movesList[0].lrPosition := 10;
PERS.recipeList[0].linearAxis[LinearAxis_e.ST130_10Z].movesList[1].lrPosition := 50;

// ST145
PERS.recipeList[0].linearAxis[LinearAxis_e.ST145_01Y].movesList[0].lrPosition := 10;
PERS.recipeList[0].linearAxis[LinearAxis_e.ST145_01Y].movesList[1].lrPosition := 100;

PERS.recipeList[0].linearAxis[LinearAxis_e.ST145_02Z].movesList[0].lrPosition := 10;
PERS.recipeList[0].linearAxis[LinearAxis_e.ST145_02Z].movesList[1].lrPosition := 50;
PERS.recipeList[0].linearAxis[LinearAxis_e.ST145_02Z].movesList[2].lrPosition := 2;
PERS.recipeList[0].linearAxis[LinearAxis_e.ST145_02Z].movesList[3].lrPosition := 50;
PERS.recipeList[0].linearAxis[LinearAxis_e.ST145_02Z].movesList[4].lrPosition := 80;

// ST180
PERS.recipeList[0].linearAxis[LinearAxis_e.ST180_01Y].movesList[0].lrPosition := 10;
PERS.recipeList[0].linearAxis[LinearAxis_e.ST180_01Y].movesList[1].lrPosition := 100;

PERS.recipeList[0].linearAxis[LinearAxis_e.ST180_02Z].movesList[0].lrPosition := 10;
PERS.recipeList[0].linearAxis[LinearAxis_e.ST180_02Z].movesList[1].lrPosition := 50;
PERS.recipeList[0].linearAxis[LinearAxis_e.ST180_02Z].movesList[2].lrPosition := 2;
PERS.recipeList[0].linearAxis[LinearAxis_e.ST180_02Z].movesList[3].lrPosition := 50;
PERS.recipeList[0].linearAxis[LinearAxis_e.ST180_02Z].movesList[4].lrPosition := 80;

PERS.recipeList[0].linearAxis[LinearAxis_e.ST180_10Z].movesList[0].lrPosition := 10;
PERS.recipeList[0].linearAxis[LinearAxis_e.ST180_10Z].movesList[1].lrPosition := 50;

// ST185
PERS.recipeList[0].linearAxis[LinearAxis_e.ST185_01Y].movesList[0].lrPosition := 10;
PERS.recipeList[0].linearAxis[LinearAxis_e.ST185_01Y].movesList[1].lrPosition := 100;

PERS.recipeList[0].linearAxis[LinearAxis_e.ST185_02Z].movesList[0].lrPosition := 10;
PERS.recipeList[0].linearAxis[LinearAxis_e.ST185_02Z].movesList[1].lrPosition := 50;
PERS.recipeList[0].linearAxis[LinearAxis_e.ST185_02Z].movesList[2].lrPosition := 2;
PERS.recipeList[0].linearAxis[LinearAxis_e.ST185_02Z].movesList[3].lrPosition := 50;
PERS.recipeList[0].linearAxis[LinearAxis_e.ST185_02Z].movesList[4].lrPosition := 80;

PERS.recipeList[0].linearAxis[LinearAxis_e.ST185_10Z].movesList[0].lrPosition := 10;
PERS.recipeList[0].linearAxis[LinearAxis_e.ST185_10Z].movesList[1].lrPosition := 50;

// ****************************************************************************** //

// recipe ST105
PERS.recipeList[0].st105.FeederConfig.InFilterDelay := 3000;
PERS.recipeList[0].st105.FeederConfig.StartDelay    := 6000;
PERS.recipeList[0].st105.FeederConfig.StopDelay     := 6000;
PERS.recipeList[0].st105.xUseVerLeft                := TRUE;
PERS.recipeList[0].st105.xUseVerRight               := TRUE;
PERS.recipeList[0].st105.FeederSize                 := 4;
PERS.recipeList[0].st105.PickOffset_X_deci          := 0;
PERS.recipeList[0].st105.PickOffset_Y_deci          := 0;
PERS.recipeList[0].st105.PickUpPos_Z_deci           := 1500;
PERS.recipeList[0].st105.isPickOffset_X_neg         := FALSE;
PERS.recipeList[0].st105.isPickOffset_Y_neg         := FALSE;
PERS.recipeList[0].st105.isPickUpPos_Z_neg          := FALSE;

// recipe ST110
PERS.recipeList[0].st110.FeederConfig.InFilterDelay := 3000;
PERS.recipeList[0].st110.FeederConfig.StartDelay    := 6000;
PERS.recipeList[0].st110.FeederConfig.StopDelay     := 6000;
PERS.recipeList[0].st110.xUseVerLeft                := TRUE;
PERS.recipeList[0].st110.xUseVerRight               := TRUE;
PERS.recipeList[0].st110.kraft_left_raw             := 0.1;
PERS.recipeList[0].st110.kraft_right_raw            := 0.1;
PERS.recipeList[0].st110.vakum_left_pc              := 50;
PERS.recipeList[0].st110.vakum_right_pc             := 50;
PERS.recipeList[0].st110.blowPieceTof_ms            := 60;
PERS.recipeList[0].st110.waitBlowPieceTon_ms        := 60;

// recipe ST115
PERS.recipeList[0].st115.FeederConfig.InFilterDelay := 3000;
PERS.recipeList[0].st115.FeederConfig.StartDelay    := 6000;
PERS.recipeList[0].st115.FeederConfig.StopDelay     := 6000;
PERS.recipeList[0].st115.xUseVerLeft                := TRUE;
PERS.recipeList[0].st115.xUseVerRight               := TRUE;

// recipe ST120
PERS.recipeList[0].st120.FeederConfigLeft.InFilterDelay  := 3000;
PERS.recipeList[0].st120.FeederConfigLeft.StartDelay     := 6000;
PERS.recipeList[0].st120.FeederConfigLeft.StopDelay      := 6000;
PERS.recipeList[0].st120.FeederConfigRight.InFilterDelay := 3000;
PERS.recipeList[0].st120.FeederConfigRight.StartDelay    := 6000;
PERS.recipeList[0].st120.FeederConfigRight.StopDelay     := 6000;
PERS.recipeList[0].st120.xUseVerLeft                     := TRUE;
PERS.recipeList[0].st120.xUseVerRight                    := TRUE;
PERS.recipeList[0].st120.TON_PieceInSeperatorLeft        := 200;
PERS.recipeList[0].st120.TON_PieceInSeperatorRight       := 200;

// recipe ST125
PERS.recipeList[0].st125.FeederConfig.InFilterDelay := 3000;
PERS.recipeList[0].st125.FeederConfig.StartDelay    := 6000;
PERS.recipeList[0].st125.FeederConfig.StopDelay     := 6000;
PERS.recipeList[0].st125.xUseVerLeft                := TRUE;
PERS.recipeList[0].st125.xUseVerRight               := TRUE;
PERS.recipeList[0].st125.diPieceGoodMaxHeight       := 30000;
PERS.recipeList[0].st125.diPieceGoodMinHeight       := 20000;
PERS.recipeList[0].st125.diPieceWrongMaxHeight      := 20000;
PERS.recipeList[0].st125.diPieceWrongMinHeight      := 10000;

// recipe ST130
PERS.recipeList[0].st130.xUseVerLeft       := TRUE;
PERS.recipeList[0].st130.xUseVerRight      := TRUE;
PERS.recipeList[0].st130.diLoadKammer_ms   := 3000;
PERS.recipeList[0].st130.diLoadPatrone_ms  := 3000;
PERS.recipeList[0].st130.uiVibroUnderneath := 30;

// recipe ST140
PERS.recipeList[0].st140.rMaxHeightSensorLeft  := 15;
PERS.recipeList[0].st140.rMinHeightSensorLeft  := 25;
PERS.recipeList[0].st140.rMaxHeightSensorRight := 15;
PERS.recipeList[0].st140.rMinHeightSensorRight := 25;
PERS.recipeList[0].st140.xIsTypeMiniOrSmart    := TRUE;

// recipe ST145
PERS.recipeList[0].st145.FeederConfig.InFilterDelay := 3000;
PERS.recipeList[0].st145.FeederConfig.StartDelay    := 6000;
PERS.recipeList[0].st145.FeederConfig.StopDelay     := 6000;
PERS.recipeList[0].st145.xUseVerLeft                := TRUE;
PERS.recipeList[0].st145.xUseVerRight               := TRUE;

// recipe ST180
PERS.recipeList[0].st180.xUseVerLeft  := TRUE;
PERS.recipeList[0].st180.xUseVerRight := TRUE;

// recipe ST185
PERS.recipeList[0].st185.xUseVerLeft  := TRUE;
PERS.recipeList[0].st185.xUseVerRight := TRUE;

// ****************************************************************************** //

// Cylinders
FOR i := 0 TO TO_INT(StationList_e._max) - 1 BY 1 DO
    FOR ii := 0 TO CONST.MAX_CYLINDER_PER_STATION - 1 BY 1 DO
        PERS.recipeList[0].cylinder2Pos[i][ii].toAS_alarm_time := 3000;
        PERS.recipeList[0].cylinder2Pos[i][ii].toGS_alarm_time := 3000;
        PERS.recipeList[0].cylinder2Pos[i][ii].toAS_wait_time  := 0;
        PERS.recipeList[0].cylinder2Pos[i][ii].toGS_wait_time  := 0;
    END_FOR
END_FOR

END_FUNCTION

// ---- POUs/00_MAIN/_02_SAFETY.TcPOU
PROGRAM _02_SAFETY
(****************************************************************************)
//SAVETY PROGRAMM
//	04.09.2019/Dj
//
//	Version:
(****************************************************************************)
VAR
    //Module
    uiArIN_State AT %I* : ARRAY[1..7] OF UINT; //Module State 
    (* 	1=140D1 
																		2=140D3 
																		3=140D5
																		4=140D7
																		5=140D9
																		6=141D1
																		6=141D3
																		*)
    uiArOUT_State AT %I* : ARRAY[1..3] OF UINT; //Module State 
    (* 	1=141D1 
																		2=141D3 
																		3=141D5
																	*)

    //GR001 IN
    xIN_Reset_bp AT %I* : BOOL;                // blue reset button
    xArIN_Input1 AT %I* : ARRAY[0..7] OF BOOL; //Mapping Inputs 
    xArIN_Input2 AT %I* : ARRAY[0..7] OF BOOL; //Mapping Inputs 
    xArIN_Input3 AT %I* : ARRAY[0..7] OF BOOL; //Mapping Inputs 
    xArIN_Input4 AT %I* : ARRAY[0..7] OF BOOL; //Mapping Inputs 
    xArIN_Input5 AT %I* : ARRAY[0..7] OF BOOL; //Mapping Inputs 
    xArIN_Input6 AT %I* : ARRAY[0..7] OF BOOL; //Mapping Inputs 
    xArIN_Input7 AT %I* : ARRAY[0..7] OF BOOL; //Mapping Inputs 
    (* 	1=140D1 
																		2=140D3 
																		3=140D5
																		4=140D7
																		5=140D9
																		6=141D1
																		7=141D3
																	*)
    //GR002 EStop						
    xIN_ESdelOut AT %I* : BOOL; //EStop del Out
    xIN_ESout    AT %I* : BOOL; //EStop	Out
    xOUT_ResetES AT %Q* : BOOL; //Reset ES

    //GR003 Türen
    xIN_MonDelOut AT %I* : BOOL; //Mon del Out Türen
    xIN_MonOut    AT %I* : BOOL; //Mon Out Türen

    //GR004 AXIS

    //GR005 OUT

    //FB's
    _FB_Gr001Input   : FB_Safety;
    _FB_Gr002NotHalt : FB_Safety;
    _FB_Gr003Tuer    : FB_Safety;
    _FB_Gr004Axis    : FB_Safety;
    _FB_Gr005Output  : FB_Safety;
    _FB_Gr010InputB  : FB_Safety;

END_VAR
VAR_OUTPUT
    xOUT_MonDelOut : BOOL; //Mon del Out
    xOUT_MonOut    : BOOL; //Mon Out	

    xOUT_ESdelOut : BOOL; //EStop del Out
    xOUT_ESout    : BOOL; //EStop Out	

    xOUT_SafetyError     : BOOL; //Error Safety
    xOUT_NotAusBetaetigt : BOOL; //Kein Not-Aus gedrückt
    xOUT_Einrichten      : BOOL; //Einrichten -1-

    XOUT_ST1 : BOOL; //Türe1
    XOUT_ST2 : BOOL; //Türe2
    XOUT_HTA : BOOL; //HubtürA
    XOUT_HTB : BOOL; //HubtürB
    XOUT_HTC : BOOL; //HubtürC
    XOUT_HTD : BOOL; //HubtürD

    XOUT_ESA : BOOL; //NOT-AUS A
    XOUT_ESB : BOOL; //NOT-AUS B
    XOUT_ESC : BOOL; //NOT-AUS C
    XOUT_ESD : BOOL; //NOT-AUS D
    XOUT_ESH : BOOL; //NOT-AUS H
    XOUT_ESP : BOOL; //NOT-AUS Panel
END_VAR

//--------------------------------------------------------------------------
//SAFETY BAUSTEINE AUFRUFEN
//--------------------------------------------------------------------------	
_FB_Gr001Input(tIN_ResetTime := T#500MS);
_FB_Gr002NotHalt(tIN_ResetTime := T#500MS);
_FB_Gr003Tuer(tIN_ResetTime := T#500MS);
_FB_Gr004Axis(tIN_ResetTime := T#500MS);
_FB_Gr005Output(tIN_ResetTime := T#500MS);
_FB_Gr010InputB(tIN_ResetTime := T#500MS);

//BAUSTEIN ERROR
xOUT_SafetyError := _FB_Gr001Input.xIN_ComErr OR //Gruppe Input
                    _FB_Gr001Input.xIN_FBErr OR
                    _FB_Gr001Input.xIN_OtherErr OR
                    _FB_Gr002NotHalt.xIN_ComErr OR //Gruppe Not-Halt
                    _FB_Gr002NotHalt.xIN_FBErr OR
                    _FB_Gr002NotHalt.xIN_OtherErr OR
                    _FB_Gr003Tuer.xIN_ComErr OR //Gruppe Tür
                    _FB_Gr003Tuer.xIN_FBErr OR
                    _FB_Gr003Tuer.xIN_OtherErr OR
                    _FB_Gr004Axis.xIN_ComErr OR //Gruppe Achsen
                    _FB_Gr004Axis.xIN_FBErr OR
                    _FB_Gr004Axis.xIN_OtherErr OR
                    _FB_Gr005Output.xIN_ComErr OR //Gruppe Output
                    _FB_Gr005Output.xIN_FBErr OR
                    _FB_Gr005Output.xIN_OtherErr OR
                    _FB_Gr001Input.xIN_ComErr OR //Gruppe InputB
                    _FB_Gr001Input.xIN_FBErr OR
                    _FB_Gr001Input.xIN_OtherErr;

//--------------------------------------------------------------------------
//NOT-AUS / ENERGIE ZUUSAMMENFASSUNG
//--------------------------------------------------------------------------	
xOUT_ESdelOut := xIN_ESdelOut;
xOUT_ESOut    := xIN_ESOut;

xOUT_MonDelOut := xIN_MonDelOut;
xOUT_MonOut    := xIN_MonOut;

//--------------------------------------------------------------------------
//NOT-AUS - TÜREN für HMI, TASTEN NICHT ENTRIEGELT	
//--------------------------------------------------------------------------	
//XOUT_ST1 := xArIN_Input5[0] AND xArIN_Input5[1]; //Türe1
//XOUT_ST2 := xArIN_Input5[2] AND
//            xArIN_Input5[3] AND
//            xArIN_Input5[4] AND
//            xArIN_Input5[5]; //Türe2

//XOUT_HTA := xArIN_Input6[0] AND xArIN_Input6[1]; //Hubtüre A
//XOUT_HTB := xArIN_Input6[2] AND xArIN_Input6[3]; //Hubtüre B
//XOUT_HTC := xArIN_Input6[4] AND xArIN_Input6[5]; //Hubtüre C
//XOUT_HTD := xArIN_Input6[6] AND xArIN_Input6[7]; //Hubtüre D
//
//XOUT_ESA := xArIN_Input1[0] AND xArIN_Input1[1]; //NOT-AUS A
//XOUT_ESB := xArIN_Input1[2] AND xArIN_Input1[3]; //NOT-AUS A
//XOUT_ESC := xArIN_Input1[4] AND xArIN_Input1[5]; //NOT-AUS A
//XOUT_ESD := xArIN_Input1[6] AND xArIN_Input1[7]; //NOT-AUS A
//XOUT_ESH := xArIN_Input2[6] AND xArIN_Input2[7]; //NOT-AUS A
//XOUT_ESP := xArIN_Input3[2] AND xArIN_Input3[3]; //NOT-AUS A
//
//xOUT_NotAusBetaetigt := XOUT_ESA AND
//                        XOUT_ESB AND
//                        XOUT_ESC AND
//                        XOUT_ESD AND
//                        XOUT_ESH AND
//                        XOUT_ESP;

//--------------------------------------------------------------------------
//RESET + Einrichten	
//--------------------------------------------------------------------------
xOUT_ResetES    := HMI.Tast_BL OR IN.I_CPX9_1_ResetBp;
xOUT_Einrichten := xArIN_Input3[1];

////--------------------------------------------------------------------------
////Tür Verriegelung	
////--------------------------------------------------------------------------
//// OUT.Q020_T1_VERR  := (HMI.enState > enState.StateSTEP);
//// OUT.Q021_T2L_VERR := OUT.Q020_T1_VERR;
//// OUT.Q022_T2R_VERR := OUT.Q020_T1_VERR;
//
//xOUT_ESout     := TRUE;
//xOUT_ESdelOut  := TRUE;
//xOUT_MonOut    := TRUE;
//xOUT_MonDelOut := TRUE;
//xOUT_Einrichten := FALSE;  // true when doors are open

END_PROGRAM

// ---- POUs/10_HMI/_10_HMI.TcPOU
PROGRAM _10_HMI
(****************************************************************************)
//HMI PROGRAMM
//	- HMI RELEVANTE Signale und Funktionen
//
//	04.09.2019/Dj
//
//	Version:
(****************************************************************************)

VAR
    //Startup HMI-Panel
    TON_startup     : TON;
    fb_startProcess : NT_StartProcess;

    //Reset Counter
    TON_ResetCounter : TON; // Reset Temparary Counter

    //Ticker
    TICK6M      : TP; // Ticker for Operating Hours
    TICK6M_     : TP;
    x_TICK6M    : BOOL;
    BLINK_500   : TP; // Ticker for Operating Hours
    BLINK_500_  : TP;
    x_BLINK_500 : BOOL;

    BLINK_100   : TP; // Ticker for Operating Hours
    BLINK_100_  : TP;
    x_BLINK_100 : BOOL;

    //Cycle Time
    _FB_SystemTime : GETSYSTEMTIME;
    dw_ActTime     : DWORD;

    //Lampen
    _FB_LAMPE : FB_LampeBNI007F;

    // keba keys
    _key_keba_1    : FB_Keba_key;
    _key_keba_2    : FB_Keba_key;
    _key_press_tof : TOF;

    // pers variable save
    _fb_bp_pers_save      : FB_BUTTON;
    fbWritePersistentData : WritePersistentData;

    //Alarmlog
    iCount6h : INT;    //6h Ticker (für AlarmLOG)
    rtNOTAUS : R_TRIG; //Trigger 6h	

    //Divers
    idx        : INT; //Index
    _12_HMI_BT : FB_HMI_BT;

    iJogValueIndex : INT := 4; // index used to know current jog velocty from lookup table
END_VAR

//***********************************************************************************************)
//Startup Terminal
//***********************************************************************************************)
TON_Startup(IN := TRUE, PT := T#5S);
fb_startProcess(NETID     := '',
                PATHSTR   := 'C:\Program Files (x86)\SpiderControl\MicroBrowser\MicroBrowser_XP.exe',
                DIRNAME   := 'C:\Users\Administrator\AppData\Roaming\SpiderControl\Microbrowser',
                COMNDLINE :=,
                START     := TON_Startup.Q,
                TMOUT     := T#10S);

//***********************************************************************************************)
//Parameter ÜBERPRÜFEN
//***********************************************************************************************)
_11_PAR_CHK();

//***********************************************************************************************)
// HMI BP
//***********************************************************************************************)
_12_HMI_BT();
_key_keba_1(s_in :=); // s_in is set by the keba panel 1 (ST105 - ST155)
_key_keba_2(s_in :=); // s_in is set by the keba panel 1 (ST160 - ST185)

IF (_key_keba_1.F12.press OR _key_keba_2.F12.press) AND (iJogValueIndex > 0) AND NOT _key_press_tof.Q THEN
    iJogValueIndex := iJogValueIndex - 1;

ELSIF (_key_keba_1.F11.press OR _key_keba_2.F11.press) AND (iJogValueIndex < 7) AND NOT _key_press_tof.Q
    THEN
    iJogValueIndex := iJogValueIndex + 1;
END_IF

AXIS.rJogVelo_pc := AXIS.arrJogValues[iJogValueIndex];

// this needs to be placed below the rJogVelo_pc management
_key_press_tof(IN := (_key_keba_1.F11.press OR
                     _key_keba_2.F11.press OR
                     _key_keba_1.F12.press OR
                     _key_keba_2.F12.press) AND
                     NOT _key_press_tof.Q,
               PT := DINT_TO_TIME(500 *
                                  TO_DINT(_key_keba_1.F11.press OR // set time to 0
                                          _key_keba_2.F11.press OR // when no key is
                                          _key_keba_1.F12.press OR // pressed
                                          _key_keba_2.F12.press)));

_fb_bp_pers_save(pbtIN  := ADR(HMI.btWritePers),
                 xINdis := FALSE,
                 xINon  := fbWritePersistentData.BUSY,
                 xINerr := fbWritePersistentData.ERR);

fbWritePersistentData(NETID := '',
                      PORT  := 851,
                      START := HMI.btWritePers.rtrig,
                      TMOUT := T#1S);

//***********************************************************************************************)
//State
//***********************************************************************************************)
_14_STATE();

//***********************************************************************************************)
//Lampen
//***********************************************************************************************)
_FB_LAMPE(enIN_State         := HMI.enState,
          xIN_AlarmAktiv     := GVL.st105_aut.xOUT_AlarmST,
          xIN_SafetyError    := _02_Safety.xOUT_SafetyError,
          xIN_NotAus         := _02_Safety.xOUT_NotAusBetaetigt,
          xIN_Mel_1_GN_GN_YE :=,
          xIN_Mel_2_GN_YE_GN :=,
          xIN_Mel_3_GN_YE_YE :=,
          xIN_Mel_4_YE_GN_GN :=,
          xIN_Mel_5_YE_GN_YE :=,
          xIN_Mel_6_YE_YE_GN :=,
          xIN_Mel_7_YE_YE_YE :=,
          tIN_Meldungen      := T#1000MS,
          tIN_Impuls         := T#500ms,
          xOUT_ErrFlag       =>);

// BALLUFF LAMPE
IO_BOX.Q0000_Balluf_Lampe_1_word     := _FB_LAMPE.wOUT_Lampe;
IO_BOX.Q5000_Balluf_Lampe_2_word     := _FB_LAMPE.wOUT_Lampe;
IO_BOX.Q0001_Balluf_Lampe_1_SycStart := _FB_LAMPE.xOUT_SyncStart;
IO_BOX.Q5001_Balluf_Lampe_2_SycStart := _FB_LAMPE.xOUT_SyncStart;
IO_BOX.Q0002_Balluf_Lampe_1_SycImp   := _FB_LAMPE.xOUT_SyncImp;
IO_BOX.Q5002_Balluf_Lampe_2_SycImp   := _FB_LAMPE.xOUT_SyncImp;

//LAMPE ENERGIE EIN 
(*
OUT.Q000_LAMP_NRJ:= _10_HMI.x_BLINK_500 AND 
						//Notaus Schalter
						_02_Safety.bArIN_Input[1].4 AND
						_02_Safety.bArIN_Input[2].0 AND	
						_02_Safety.bArIN_Input[2].2 AND
						_02_Safety.bArIN_Input[2].4 AND
						_02_Safety.bArIN_Input[2].6 
					OR (HMI.enState>enState.StateOFF);
					*)

OUT.Q_CPX9_1_EnergiEin_led   := _02_SAFETY.xOUT_ESout;
OUT.Q_CPX9_1_Process_running := HMI.enState > enState.StateSTOP OR HMI.enState = enState.StateREADY;
OUT.Q_CPX9_1_Process_stopped := HMI.enState <= enState.StateSTOP;

